LIN {X 0,Y 260.477,Z 576.066,A -85,B 0,C 180,E1 -18837.737,E2 -18837.737} C_VEL
LIN {X 0,Y 264.246,Z 563.841,A -85,B 0,C 180,E1 -18840.132,E2 -18840.132} C_VEL
LIN {X 0,Y 267.827,Z 551.379,A -85,B 0,C 180,E1 -18842.097,E2 -18842.097} C_VEL
LIN {X 0,Y 271.196,Z 538.149,A -85,B 0,C 180,E1 -18843.781,E2 -18843.781} C_VEL
LIN {X 0,Y 274.264,Z 524.044,A -85,B 0,C 180,E1 -18845.208,E2 -18845.208} C_VEL
LIN {X 0,Y 276.82,Z 510.254,A -85,B 0,C 180,E1 -18846.288,E2 -18846.288} C_VEL
LIN {X 0,Y 279.114,Z 494.819,A -85,B 0,C 180,E1 -18847.178,E2 -18847.178} C_VEL
LIN {X 0,Y 280.649,Z 479.547,A -85,B 0,C 180,E1 -18847.787,E2 -18847.787} C_VEL
LIN {X 0,Y 285.626,Z 378.515,A -85,B 0,C 180,E1 -18850.247,E2 -18850.247} C_VEL
LIN {X 0,Y 285.487,Z 376.742,A -85,B 0,C 180,E1 -18850.327,E2 -18850.327} C_VEL
LIN {X 0,Y 278.337,Z 360.16,A -85,B 0,C 180,E1 -18852.139,E2 -18852.139} C_VEL
LIN {X 0,Y 270.765,Z 345.131,A -85,B 0,C 180,E1 -18854.134,E2 -18854.134} C_VEL
LIN {X 0,Y 263.382,Z 332.001,A -85,B 0,C 180,E1 -18856.203,E2 -18856.203} C_VEL
LIN {X 0,Y 256.795,Z 321.549,A -85,B 0,C 180,E1 -18858.171,E2 -18858.171} C_VEL
LIN {X 0,Y 253.581,Z 316.573,A -85,B 0,C 180,E1 -18859.193,E2 -18859.193} C_VEL
LIN {X 0,Y 250.484,Z 311.706,A -85,B 0,C 180,E1 -18860.269,E2 -18860.269} C_VEL
LIN {X 0,Y 249.039,Z 307.085,A -85,B 0,C 180,E1 -18862.618,E2 -18862.618} C_VEL
LIN {X 0,Y 249.037,Z 307.088,A -85,B 0,C 180,E1 -18865.639,E2 -18865.639} C_VEL
LIN {X 0,Y 248.994,Z 307.089,A -85,B 0,C 180,E1 -18869.465,E2 -18869.465} C_VEL
LIN {X 0,Y 249.008,Z 307.086,A -85,B 0,C 180,E1 -18873.155,E2 -18873.155} C_VEL
LIN {X 0,Y 248.998,Z 307.089,A -85,B 0,C 180,E1 -18876.725,E2 -18876.725} C_VEL
LIN {X 0,Y 249.038,Z 307.057,A -85,B 0,C 180,E1 -18880.206,E2 -18880.206} C_VEL
LIN {X 0,Y 249.151,Z 307.067,A -85,B 0,C 180,E1 -18883.616,E2 -18883.616} C_VEL
LIN {X 0,Y 249.177,Z 307.04,A -85,B 0,C 180,E1 -18886.96,E2 -18886.96} C_VEL
LIN {X 0,Y 249.365,Z 307.025,A -85,B 0,C 180,E1 -18890.538,E2 -18890.538} C_VEL
LIN {X 0,Y 249.415,Z 307.035,A -85,B 0,C 180,E1 -18893.529,E2 -18893.529} C_VEL
LIN {X 0,Y 249.653,Z 307.001,A -85,B 0,C 180,E1 -18898.387,E2 -18898.387} C_VEL
LIN {X 0,Y 249.65,Z 307.007,A -85,B 0,C 180,E1 -18901.613,E2 -18901.613} C_VEL
LIN {X 0,Y 249.416,Z 307.032,A -85,B 0,C 180,E1 -18906.679,E2 -18906.679} C_VEL
LIN {X 0,Y 249.326,Z 307.05,A -85,B 0,C 180,E1 -18909.737,E2 -18909.737} C_VEL
LIN {X 0,Y 249.164,Z 307.065,A -85,B 0,C 180,E1 -18914.706,E2 -18914.706} C_VEL
LIN {X 0,Y 249.088,Z 307.072,A -85,B 0,C 180,E1 -18918.081,E2 -18918.081} C_VEL
LIN {X 0,Y 249.041,Z 307.055,A -85,B 0,C 180,E1 -18921.523,E2 -18921.523} C_VEL
LIN {X 0,Y 249.107,Z 307.067,A -85,B 0,C 180,E1 -18925.474,E2 -18925.474} C_VEL
LIN {X 0,Y 249.058,Z 307.066,A -85,B 0,C 180,E1 -18928.986,E2 -18928.986} C_VEL
LIN {X 0,Y 249.026,Z 307.084,A -85,B 0,C 180,E1 -18932.427,E2 -18932.427} C_VEL
LIN {X 0,Y 249.043,Z 307.088,A -85,B 0,C 180,E1 -18936.343,E2 -18936.343} C_VEL
LIN {X 0,Y 249.022,Z 307.166,A -85,B 0,C 180,E1 -18939.617,E2 -18939.617} C_VEL
LIN {X 0,Y 249.906,Z 309.755,A -85,B 0,C 180,E1 -18939.977,E2 -18939.977} C_VEL
LIN {X 0,Y 251.813,Z 311.92,A -85,B 0,C 180,E1 -18940.59,E2 -18940.59} C_VEL
LIN {X 0,Y 252.602,Z 312.645,A -85,B 0,C 180,E1 -18940.831,E2 -18940.831} C_VEL
LIN {X 0,Y 254.745,Z 315.993,A -85,B 0,C 180,E1 -18941.53,E2 -18941.53} C_VEL
LIN {X 0,Y 256.163,Z 317.683,A -85,B 0,C 180,E1 -18941.96,E2 -18941.96} C_VEL
LIN {X 0,Y 258.928,Z 321.433,A -85,B 0,C 180,E1 -18942.792,E2 -18942.792} C_VEL
LIN {X 0,Y 268.098,Z 334.977,A -85,B 0,C 180,E1 -18945.388,E2 -18945.388} C_VEL
LIN {X 0,Y 274.88,Z 345.917,A -85,B 0,C 180,E1 -18947.161,E2 -18947.161} C_VEL
LIN {X 0,Y 281.793,Z 359.713,A -85,B 0,C 180,E1 -18948.921,E2 -18948.921} C_VEL
LIN {X 0,Y 285.944,Z 368.841,A -85,B 0,C 180,E1 -18949.943,E2 -18949.943} C_VEL
LIN {X 0,Y 281.179,Z 467.093,A -85,B 0,C 180,E1 -18952.353,E2 -18952.353} C_VEL
LIN {X 0,Y 279.682,Z 482.247,A -85,B 0,C 180,E1 -18952.967,E2 -18952.967} C_VEL
LIN {X 0,Y 277.739,Z 496.979,A -85,B 0,C 180,E1 -18953.851,E2 -18953.851} C_VEL
LIN {X 0,Y 275.33,Z 511.361,A -85,B 0,C 180,E1 -18955.013,E2 -18955.013} C_VEL
LIN {X 0,Y 272.275,Z 525.892,A -85,B 0,C 180,E1 -18956.515,E2 -18956.515} C_VEL
LIN {X 0,Y 269.174,Z 538.098,A -85,B 0,C 180,E1 -18958.082,E2 -18958.082} C_VEL
LIN {X 0,Y 266.055,Z 549.441,A -85,B 0,C 180,E1 -18959.875,E2 -18959.875} C_VEL
LIN {X 0,Y 262.464,Z 561.007,A -85,B 0,C 180,E1 -18962.085,E2 -18962.085} C_VEL
LIN {X 0,Y 259.548,Z 570.521,A -85,B 0,C 180,E1 -18964.327,E2 -18964.327} C_VEL
LIN {X 0,Y 256.366,Z 579.961,A -85,B 0,C 180,E1 -18967.006,E2 -18967.006} C_VEL
LIN {X 0,Y 253.642,Z 587.816,A -85,B 0,C 180,E1 -18969.736,E2 -18969.736} C_VEL
LIN {X 0,Y 251.256,Z 595.141,A -85,B 0,C 180,E1 -18972.921,E2 -18972.921} C_VEL
LIN {X 0,Y 249.39,Z 600.95,A -85,B 0,C 180,E1 -18976.141,E2 -18976.141} C_VEL
LIN {X 0,Y 248.47,Z 604.384,A -85,B 0,C 180,E1 -18978.581,E2 -18978.581} C_VEL
LIN {X 0,Y 247.638,Z 607.86,A -85,B 0,C 180,E1 -18981.842,E2 -18981.842} C_VEL
LIN {X 0,Y 247.134,Z 610.155,A -85,B 0,C 180,E1 -18985.106,E2 -18985.106} C_VEL
LIN {X 0,Y 246.995,Z 611.323,A -85,B 0,C 180,E1 -18988.37,E2 -18988.37} C_VEL
LIN {X 0,Y 246.994,Z 611.336,A -85,B 0,C 180,E1 -18991.63,E2 -18991.63} C_VEL
LIN {X 0,Y 247.128,Z 610.22,A -85,B 0,C 180,E1 -18994.894,E2 -18994.894} C_VEL
LIN {X 0,Y 247.576,Z 607.975,A -85,B 0,C 180,E1 -18998.16,E2 -18998.16} C_VEL
LIN {X 0,Y 248.443,Z 604.544,A -85,B 0,C 180,E1 -19001.421,E2 -19001.421} C_VEL
LIN {X 0,Y 249.783,Z 599.845,A -85,B 0,C 180,E1 -19004.668,E2 -19004.668} C_VEL
LIN {X 0,Y 251.755,Z 593.749,A -85,B 0,C 180,E1 -19007.883,E2 -19007.883} C_VEL
LIN {X 0,Y 254.327,Z 586.069,A -85,B 0,C 180,E1 -19011.053,E2 -19011.053} C_VEL
LIN {X 0,Y 257.145,Z 577.876,A -85,B 0,C 180,E1 -19013.773,E2 -19013.773} C_VEL
LIN {X 0,Y 260.504,Z 567.999,A -85,B 0,C 180,E1 -19016.432,E2 -19016.432} C_VEL
LIN {X 0,Y 263.554,Z 557.877,A -85,B 0,C 180,E1 -19018.684,E2 -19018.684} C_VEL
LIN {X 0,Y 267.19,Z 545.809,A -85,B 0,C 180,E1 -19020.857,E2 -19020.857} C_VEL
LIN {X 0,Y 270.434,Z 533.706,A -85,B 0,C 180,E1 -19022.631,E2 -19022.631} C_VEL
LIN {X 0,Y 273.51,Z 520.55,A -85,B 0,C 180,E1 -19024.199,E2 -19024.199} C_VEL
LIN {X 0,Y 276.065,Z 507.506,A -85,B 0,C 180,E1 -19025.447,E2 -19025.447} C_VEL
LIN {X 0,Y 278.318,Z 493.311,A -85,B 0,C 180,E1 -19026.511,E2 -19026.511} C_VEL
LIN {X 0,Y 280.218,Z 478.014,A -85,B 0,C 180,E1 -19027.345,E2 -19027.345} C_VEL
LIN {X 0,Y 281.501,Z 463.213,A -85,B 0,C 180,E1 -19027.879,E2 -19027.879} C_VEL
LIN {X 0,Y 286.04,Z 368.931,A -85,B 0,C 180,E1 -19030.172,E2 -19030.172} C_VEL
LIN {X 0,Y 278.222,Z 352.196,A -85,B 0,C 180,E1 -19032.124,E2 -19032.124} C_VEL
LIN {X 0,Y 273.365,Z 343.191,A -85,B 0,C 180,E1 -19033.376,E2 -19033.376} C_VEL
LIN {X 0,Y 265.536,Z 331.06,A -85,B 0,C 180,E1 -19035.462,E2 -19035.462} C_VEL
LIN {X 0,Y 258.345,Z 320.791,A -85,B 0,C 180,E1 -19037.531,E2 -19037.531} C_VEL
LIN {X 0,Y 255.483,Z 316.712,A -85,B 0,C 180,E1 -19038.412,E2 -19038.412} C_VEL
LIN {X 0,Y 253.02,Z 313.492,A -85,B 0,C 180,E1 -19039.185,E2 -19039.185} C_VEL
LIN {X 0,Y 252.146,Z 312.144,A -85,B 0,C 180,E1 -19039.475,E2 -19039.475} C_VEL
LIN {X 0,Y 250.089,Z 310.064,A -85,B 0,C 180,E1 -19040.125,E2 -19040.125} C_VEL
LIN {X 0,Y 249.079,Z 307.384,A -85,B 0,C 180,E1 -19040.525,E2 -19040.525} C_VEL
LIN {X 0,Y 249.015,Z 307.093,A -85,B 0,C 180,E1 -19040.578,E2 -19040.578} C_VEL
LIN {X 0,Y 249.039,Z 307.073,A -85,B 0,C 180,E1 -19044.922,E2 -19044.922} C_VEL
LIN {X 0,Y 249.001,Z 307.059,A -85,B 0,C 180,E1 -19049.466,E2 -19049.466} C_VEL
LIN {X 0,Y 249.053,Z 307.086,A -85,B 0,C 180,E1 -19053.16,E2 -19053.16} C_VEL
LIN {X 0,Y 249.052,Z 307.087,A -85,B 0,C 180,E1 -19056.73,E2 -19056.73} C_VEL
LIN {X 0,Y 249.077,Z 307.084,A -85,B 0,C 180,E1 -19060.209,E2 -19060.209} C_VEL
LIN {X 0,Y 249.097,Z 307.071,A -85,B 0,C 180,E1 -19061.859,E2 -19061.859} C_VEL
LIN {X 0,Y 248.501,Z 307.151,A -85,B 0,C 180,E1 -19063.21,E2 -19063.21} C_VEL
LIN {X 0,Y 245.667,Z 307.506,A -85,B 0,C 180,E1 -19065.413,E2 -19065.413} C_VEL
LIN {X 0,Y 243.243,Z 307.808,A -85,B 0,C 180,E1 -19067.207,E2 -19067.207} C_VEL
LIN {X 0,Y 242.239,Z 307.936,A -85,B 0,C 180,E1 -19068.6,E2 -19068.6} C_VEL
LIN {X 0,Y 242.18,Z 307.936,A -85,B 0,C 180,E1 -19069.072,E2 -19069.072} C_VEL
LIN {X 0,Y 242.382,Z 307.907,A -85,B 0,C 180,E1 -19071.664,E2 -19071.664} C_VEL
LIN {X 0,Y 242.226,Z 307.925,A -85,B 0,C 180,E1 -19075.006,E2 -19075.006} C_VEL
LIN {X 0,Y 242.617,Z 307.888,A -85,B 0,C 180,E1 -19078.34,E2 -19078.34} C_VEL
LIN {X 0,Y 242.613,Z 307.887,A -85,B 0,C 180,E1 -19081.66,E2 -19081.66} C_VEL
LIN {X 0,Y 242.397,Z 307.917,A -85,B 0,C 180,E1 -19086.66,E2 -19086.66} C_VEL
LIN {X 0,Y 242.259,Z 307.925,A -85,B 0,C 180,E1 -19090.024,E2 -19090.024} C_VEL
LIN {X 0,Y 242.114,Z 307.952,A -85,B 0,C 180,E1 -19095.144,E2 -19095.144} C_VEL
LIN {X 0,Y 242.024,Z 307.956,A -85,B 0,C 180,E1 -19098.628,E2 -19098.628} C_VEL
LIN {X 0,Y 241.967,Z 307.961,A -85,B 0,C 180,E1 -19102.184,E2 -19102.184} C_VEL
LIN {X 0,Y 241.981,Z 307.959,A -85,B 0,C 180,E1 -19105.827,E2 -19105.827} C_VEL
LIN {X 0,Y 241.962,Z 307.972,A -85,B 0,C 180,E1 -19109.589,E2 -19109.589} C_VEL
LIN {X 0,Y 241.974,Z 307.959,A -85,B 0,C 180,E1 -19113.493,E2 -19113.493} C_VEL
LIN {X 0,Y 241.998,Z 308.143,A -85,B 0,C 180,E1 -19115.739,E2 -19115.739} C_VEL
LIN {X 0,Y 243.266,Z 311.805,A -85,B 0,C 180,E1 -19117.623,E2 -19117.623} C_VEL
LIN {X 0,Y 246.159,Z 316.163,A -85,B 0,C 180,E1 -19118.682,E2 -19118.682} C_VEL
LIN {X 0,Y 248.289,Z 319.312,A -85,B 0,C 180,E1 -19119.428,E2 -19119.428} C_VEL
LIN {X 0,Y 251.893,Z 324.806,A -85,B 0,C 180,E1 -19120.644,E2 -19120.644} C_VEL
LIN {X 0,Y 257.896,Z 334.42,A -85,B 0,C 180,E1 -19122.552,E2 -19122.552} C_VEL
LIN {X 0,Y 265.153,Z 347.057,A -85,B 0,C 180,E1 -19124.701,E2 -19124.701} C_VEL
LIN {X 0,Y 272.745,Z 362.134,A -85,B 0,C 180,E1 -19126.815,E2 -19126.815} C_VEL
LIN {X 0,Y 279.117,Z 376.624,A -85,B 0,C 180,E1 -19128.511,E2 -19128.511} C_VEL
LIN {X 0,Y 280.222,Z 379.318,A -85,B 0,C 180,E1 -19128.799,E2 -19128.799} C_VEL
LIN {X 0,Y 275.522,Z 474.523,A -85,B 0,C 180,E1 -19131.148,E2 -19131.148} C_VEL
LIN {X 0,Y 274.146,Z 489.815,A -85,B 0,C 180,E1 -19131.68,E2 -19131.68} C_VEL
LIN {X 0,Y 271.984,Z 505.365,A -85,B 0,C 180,E1 -19132.495,E2 -19132.495} C_VEL
LIN {X 0,Y 269.297,Z 520.239,A -85,B 0,C 180,E1 -19133.58,E2 -19133.58} C_VEL
LIN {X 0,Y 266.114,Z 534.597,A -85,B 0,C 180,E1 -19134.955,E2 -19134.955} C_VEL
LIN {X 0,Y 262.902,Z 547.521,A -85,B 0,C 180,E1 -19136.541,E2 -19136.541} C_VEL
LIN {X 0,Y 259.416,Z 559.534,A -85,B 0,C 180,E1 -19138.339,E2 -19138.339} C_VEL
LIN {X 0,Y 255.899,Z 570.666,A -85,B 0,C 180,E1 -19140.374,E2 -19140.374} C_VEL
LIN {X 0,Y 252.446,Z 581.236,A -85,B 0,C 180,E1 -19142.745,E2 -19142.745} C_VEL
LIN {X 0,Y 249.249,Z 590.949,A -85,B 0,C 180,E1 -19145.425,E2 -19145.425} C_VEL
LIN {X 0,Y 246.294,Z 599.278,A -85,B 0,C 180,E1 -19148.226,E2 -19148.226} C_VEL
LIN {X 0,Y 243.714,Z 607.112,A -85,B 0,C 180,E1 -19151.506,E2 -19151.506} C_VEL
LIN {X 0,Y 241.837,Z 613.352,A -85,B 0,C 180,E1 -19154.839,E2 -19154.839} C_VEL
LIN {X 0,Y 240.593,Z 618.183,A -85,B 0,C 180,E1 -19158.201,E2 -19158.201} C_VEL
LIN {X 0,Y 239.985,Z 621.73,A -85,B 0,C 180,E1 -19161.58,E2 -19161.58} C_VEL
LIN {X 0,Y 239.765,Z 624.067,A -85,B 0,C 180,E1 -19164.955,E2 -19164.955} C_VEL
LIN {X 0,Y 239.829,Z 625.244,A -85,B 0,C 180,E1 -19168.321,E2 -19168.321} C_VEL
LIN {X 0,Y 239.89,Z 625.4,A -85,B 0,C 180,E1 -19170,E2 -19170} C_VEL
LIN {X 0,Y 239.744,Z 624.785,A -85,B 0,C 180,E1 -19173.361,E2 -19173.361} C_VEL
LIN {X 0,Y 239.785,Z 623.015,A -85,B 0,C 180,E1 -19176.733,E2 -19176.733} C_VEL
LIN {X 0,Y 240.229,Z 620.071,A -85,B 0,C 180,E1 -19180.109,E2 -19180.109} C_VEL
LIN {X 0,Y 241.167,Z 615.885,A -85,B 0,C 180,E1 -19183.481,E2 -19183.481} C_VEL
LIN {X 0,Y 242.591,Z 610.344,A -85,B 0,C 180,E1 -19186.84,E2 -19186.84} C_VEL
LIN {X 0,Y 244.896,Z 603.312,A -85,B 0,C 180,E1 -19190.143,E2 -19190.143} C_VEL
LIN {X 0,Y 247.899,Z 594.571,A -85,B 0,C 180,E1 -19193.384,E2 -19193.384} C_VEL
LIN {X 0,Y 250.555,Z 586.782,A -85,B 0,C 180,E1 -19195.756,E2 -19195.756} C_VEL
LIN {X 0,Y 254.146,Z 575.858,A -85,B 0,C 180,E1 -19198.49,E2 -19198.49} C_VEL
LIN {X 0,Y 258.103,Z 563.634,A -85,B 0,C 180,E1 -19200.927,E2 -19200.927} C_VEL
LIN {X 0,Y 261.445,Z 552.4,A -85,B 0,C 180,E1 -19202.75,E2 -19202.75} C_VEL
LIN {X 0,Y 265.107,Z 538.703,A -85,B 0,C 180,E1 -19204.55,E2 -19204.55} C_VEL
LIN {X 0,Y 268.472,Z 523.834,A -85,B 0,C 180,E1 -19206.085,E2 -19206.085} C_VEL
LIN {X 0,Y 271.143,Z 510.044,A -85,B 0,C 180,E1 -19207.174,E2 -19207.174} C_VEL
LIN {X 0,Y 273.5,Z 494.607,A -85,B 0,C 180,E1 -19208.075,E2 -19208.075} C_VEL
LIN {X 0,Y 275.067,Z 479.328,A -85,B 0,C 180,E1 -19208.694,E2 -19208.694} C_VEL
LIN {X 0,Y 279.58,Z 391.475,A -85,B 0,C 180,E1 -19210.864,E2 -19210.864} C_VEL
LIN {X 0,Y 280.114,Z 379.234,A -85,B 0,C 180,E1 -19211.176,E2 -19211.176} C_VEL
LIN {X 0,Y 273.524,Z 363.866,A -85,B 0,C 180,E1 -19212.921,E2 -19212.921} C_VEL
LIN {X 0,Y 266.605,Z 349.897,A -85,B 0,C 180,E1 -19214.824,E2 -19214.824} C_VEL
LIN {X 0,Y 259.318,Z 336.779,A -85,B 0,C 180,E1 -19216.951,E2 -19216.951} C_VEL
LIN {X 0,Y 253.151,Z 326.806,A -85,B 0,C 180,E1 -19218.873,E2 -19218.873} C_VEL
LIN {X 0,Y 249.75,Z 321.507,A -85,B 0,C 180,E1 -19219.997,E2 -19219.997} C_VEL
LIN {X 0,Y 246.292,Z 316.344,A -85,B 0,C 180,E1 -19221.192,E2 -19221.192} C_VEL
LIN {X 0,Y 243.196,Z 311.686,A -85,B 0,C 180,E1 -19222.319,E2 -19222.319} C_VEL
LIN {X 0,Y 241.981,Z 307.961,A -85,B 0,C 180,E1 -19224.374,E2 -19224.374} C_VEL
LIN {X 0,Y 241.947,Z 307.972,A -85,B 0,C 180,E1 -19228.476,E2 -19228.476} C_VEL
LIN {X 0,Y 241.949,Z 307.967,A -85,B 0,C 180,E1 -19232.306,E2 -19232.306} C_VEL
LIN {X 0,Y 241.95,Z 307.965,A -85,B 0,C 180,E1 -19236.005,E2 -19236.005} C_VEL
LIN {X 0,Y 241.977,Z 307.942,A -85,B 0,C 180,E1 -19239.603,E2 -19239.603} C_VEL
LIN {X 0,Y 242.107,Z 307.938,A -85,B 0,C 180,E1 -19243.318,E2 -19243.318} C_VEL
LIN {X 0,Y 242.153,Z 307.903,A -85,B 0,C 180,E1 -19248.278,E2 -19248.278} C_VEL
LIN {X 0,Y 242.351,Z 307.918,A -85,B 0,C 180,E1 -19251.663,E2 -19251.663} C_VEL
LIN {X 0,Y 242.384,Z 307.912,A -85,B 0,C 180,E1 -19253.34,E2 -19253.34} C_VEL
LIN {X 0,Y 242.612,Z 307.878,A -85,B 0,C 180,E1 -19258.34,E2 -19258.34} C_VEL
LIN {X 0,Y 242.611,Z 307.884,A -85,B 0,C 180,E1 -19261.66,E2 -19261.66} C_VEL
LIN {X 0,Y 242.398,Z 307.906,A -85,B 0,C 180,E1 -19266.66,E2 -19266.66} C_VEL
LIN {X 0,Y 242.254,Z 307.928,A -85,B 0,C 180,E1 -19270.024,E2 -19270.024} C_VEL
LIN {X 0,Y 242.114,Z 307.942,A -85,B 0,C 180,E1 -19275.144,E2 -19275.144} C_VEL
LIN {X 0,Y 242.025,Z 307.941,A -85,B 0,C 180,E1 -19278.628,E2 -19278.628} C_VEL
LIN {X 0,Y 241.983,Z 307.941,A -85,B 0,C 180,E1 -19282.183,E2 -19282.183} C_VEL
LIN {X 0,Y 242.045,Z 307.939,A -85,B 0,C 180,E1 -19285.83,E2 -19285.83} C_VEL
LIN {X 0,Y 241.999,Z 307.955,A -85,B 0,C 180,E1 -19289.585,E2 -19289.585} C_VEL
LIN {X 0,Y 241.976,Z 307.969,A -85,B 0,C 180,E1 -19293.494,E2 -19293.494} C_VEL
LIN {X 0,Y 241.988,Z 307.983,A -85,B 0,C 180,E1 -19297.582,E2 -19297.582} C_VEL
LIN {X 0,Y 242.936,Z 310.696,A -85,B 0,C 180,E1 -19298.003,E2 -19298.003} C_VEL
LIN {X 0,Y 244.853,Z 312.841,A -85,B 0,C 180,E1 -19298.677,E2 -19298.677} C_VEL
LIN {X 0,Y 245.764,Z 313.765,A -85,B 0,C 180,E1 -19298.986,E2 -19298.986} C_VEL
LIN {X 0,Y 248.012,Z 317.166,A -85,B 0,C 180,E1 -19299.78,E2 -19299.78} C_VEL
LIN {X 0,Y 249.476,Z 318.808,A -85,B 0,C 180,E1 -19300.257,E2 -19300.257} C_VEL
LIN {X 0,Y 252.072,Z 322.342,A -85,B 0,C 180,E1 -19301.105,E2 -19301.105} C_VEL
LIN {X 0,Y 259.349,Z 332.783,A -85,B 0,C 180,E1 -19303.345,E2 -19303.345} C_VEL
LIN {X 0,Y 267.478,Z 345.207,A -85,B 0,C 180,E1 -19305.635,E2 -19305.635} C_VEL
LIN {X 0,Y 272.335,Z 353.843,A -85,B 0,C 180,E1 -19306.941,E2 -19306.941} C_VEL
LIN {X 0,Y 279.378,Z 368.706,A -85,B 0,C 180,E1 -19308.787,E2 -19308.787} C_VEL
LIN {X 0,Y 280.44,Z 371.158,A -85,B 0,C 180,E1 -19309.06,E2 -19309.06} C_VEL
LIN {X 0,Y 275.6,Z 467.311,A -85,B 0,C 180,E1 -19311.453,E2 -19311.453} C_VEL
LIN {X 0,Y 274.062,Z 482.461,A -85,B 0,C 180,E1 -19312.075,E2 -19312.075} C_VEL
LIN {X 0,Y 272.049,Z 497.19,A -85,B 0,C 180,E1 -19312.97,E2 -19312.97} C_VEL
LIN {X 0,Y 269.74,Z 510.156,A -85,B 0,C 180,E1 -19314.013,E2 -19314.013} C_VEL
LIN {X 0,Y 266.756,Z 524.548,A -85,B 0,C 180,E1 -19315.499,E2 -19315.499} C_VEL
LIN {X 0,Y 263.514,Z 537.018,A -85,B 0,C 180,E1 -19317.085,E2 -19317.085} C_VEL
LIN {X 0,Y 260.264,Z 548.583,A -85,B 0,C 180,E1 -19318.907,E2 -19318.907} C_VEL
LIN {X 0,Y 256.47,Z 560.443,A -85,B 0,C 180,E1 -19321.179,E2 -19321.179} C_VEL
LIN {X 0,Y 253.169,Z 570.727,A -85,B 0,C 180,E1 -19323.631,E2 -19323.631} C_VEL
LIN {X 0,Y 249.834,Z 580.166,A -85,B 0,C 180,E1 -19326.369,E2 -19326.369} C_VEL
LIN {X 0,Y 246.978,Z 588.021,A -85,B 0,C 180,E1 -19329.164,E2 -19329.164} C_VEL
LIN {X 0,Y 244.438,Z 595.347,A -85,B 0,C 180,E1 -19332.429,E2 -19332.429} C_VEL
LIN {X 0,Y 242.477,Z 601.155,A -85,B 0,C 180,E1 -19335.738,E2 -19335.738} C_VEL
LIN {X 0,Y 241.5,Z 604.589,A -85,B 0,C 180,E1 -19338.246,E2 -19338.246} C_VEL
LIN {X 0,Y 240.61,Z 608.063,A -85,B 0,C 180,E1 -19341.602,E2 -19341.602} C_VEL
LIN {X 0,Y 240.058,Z 610.359,A -85,B 0,C 180,E1 -19344.961,E2 -19344.961} C_VEL
LIN {X 0,Y 239.907,Z 611.526,A -85,B 0,C 180,E1 -19348.321,E2 -19348.321} C_VEL
LIN {X 0,Y 239.906,Z 611.538,A -85,B 0,C 180,E1 -19351.679,E2 -19351.679} C_VEL
LIN {X 0,Y 240.058,Z 610.423,A -85,B 0,C 180,E1 -19355.039,E2 -19355.039} C_VEL
LIN {X 0,Y 240.523,Z 608.178,A -85,B 0,C 180,E1 -19358.401,E2 -19358.401} C_VEL
LIN {X 0,Y 241.458,Z 604.747,A -85,B 0,C 180,E1 -19361.756,E2 -19361.756} C_VEL
LIN {X 0,Y 242.906,Z 600.047,A -85,B 0,C 180,E1 -19365.093,E2 -19365.093} C_VEL
LIN {X 0,Y 244.989,Z 593.951,A -85,B 0,C 180,E1 -19368.394,E2 -19368.394} C_VEL
LIN {X 0,Y 247.669,Z 586.272,A -85,B 0,C 180,E1 -19371.647,E2 -19371.647} C_VEL
LIN {X 0,Y 250.646,Z 578.077,A -85,B 0,C 180,E1 -19374.429,E2 -19374.429} C_VEL
LIN {X 0,Y 254.129,Z 568.2,A -85,B 0,C 180,E1 -19377.149,E2 -19377.149} C_VEL
LIN {X 0,Y 257.328,Z 558.077,A -85,B 0,C 180,E1 -19379.445,E2 -19379.445} C_VEL
LIN {X 0,Y 261.127,Z 546.009,A -85,B 0,C 180,E1 -19381.656,E2 -19381.656} C_VEL
LIN {X 0,Y 264.492,Z 533.905,A -85,B 0,C 180,E1 -19383.459,E2 -19383.459} C_VEL
LIN {X 0,Y 267.666,Z 520.748,A -85,B 0,C 180,E1 -19385.054,E2 -19385.054} C_VEL
LIN {X 0,Y 270.175,Z 508.445,A -85,B 0,C 180,E1 -19386.255,E2 -19386.255} C_VEL
LIN {X 0,Y 272.475,Z 494.803,A -85,B 0,C 180,E1 -19387.31,E2 -19387.31} C_VEL
LIN {X 0,Y 274.44,Z 480.03,A -85,B 0,C 180,E1 -19388.155,E2 -19388.155} C_VEL
LIN {X 0,Y 275.86,Z 464.898,A -85,B 0,C 180,E1 -19388.738,E2 -19388.738} C_VEL
LIN {X 0,Y 280.557,Z 372.002,A -85,B 0,C 180,E1 -19391.028,E2 -19391.028} C_VEL
LIN {X 0,Y 280.254,Z 370.496,A -85,B 0,C 180,E1 -19391.132,E2 -19391.132} C_VEL
LIN {X 0,Y 272.656,Z 354.369,A -85,B 0,C 180,E1 -19393.12,E2 -19393.12} C_VEL
LIN {X 0,Y 267.696,Z 345.456,A -85,B 0,C 180,E1 -19394.457,E2 -19394.457} C_VEL
LIN {X 0,Y 258.168,Z 330.912,A -85,B 0,C 180,E1 -19397.166,E2 -19397.166} C_VEL
LIN {X 0,Y 251.797,Z 322.034,A -85,B 0,C 180,E1 -19399.143,E2 -19399.143} C_VEL
LIN {X 0,Y 248.627,Z 317.741,A -85,B 0,C 180,E1 -19400.19,E2 -19400.19} C_VEL
LIN {X 0,Y 246.371,Z 314.945,A -85,B 0,C 180,E1 -19400.955,E2 -19400.955} C_VEL
LIN {X 0,Y 245.408,Z 313.2,A -85,B 0,C 180,E1 -19401.315,E2 -19401.315} C_VEL
LIN {X 0,Y 243.172,Z 311.084,A -85,B 0,C 180,E1 -19402.082,E2 -19402.082} C_VEL
LIN {X 0,Y 242.041,Z 308.398,A -85,B 0,C 180,E1 -19402.558,E2 -19402.558} C_VEL
LIN {X 0,Y 241.972,Z 307.943,A -85,B 0,C 180,E1 -19402.677,E2 -19402.677} C_VEL
LIN {X 0,Y 241.983,Z 307.95,A -85,B 0,C 180,E1 -19407.377,E2 -19407.377} C_VEL
LIN {X 0,Y 241.98,Z 307.94,A -85,B 0,C 180,E1 -19410.608,E2 -19410.608} C_VEL
LIN {X 0,Y 242.045,Z 307.951,A -85,B 0,C 180,E1 -19414.18,E2 -19414.18} C_VEL
LIN {X 0,Y 242.017,Z 307.953,A -85,B 0,C 180,E1 -19418.315,E2 -19418.315} C_VEL
LIN {X 0,Y 242.11,Z 307.945,A -85,B 0,C 180,E1 -19423.316,E2 -19423.316} C_VEL
LIN {X 0,Y 242.16,Z 307.944,A -85,B 0,C 180,E1 -19428.278,E2 -19428.278} C_VEL
LIN {X 0,Y 242.18,Z 307.936,A -85,B 0,C 180,E1 -19429.072,E2 -19429.072} C_VEL
LIN {X 0,Y 241.556,Z 308.014,A -85,B 0,C 180,E1 -19430.461,E2 -19430.461} C_VEL
LIN {X 0,Y 238.684,Z 308.376,A -85,B 0,C 180,E1 -19432.726,E2 -19432.726} C_VEL
LIN {X 0,Y 236.264,Z 308.671,A -85,B 0,C 180,E1 -19434.573,E2 -19434.573} C_VEL
LIN {X 0,Y 235.3,Z 308.787,A -85,B 0,C 180,E1 -19436.007,E2 -19436.007} C_VEL
LIN {X 0,Y 235.263,Z 308.795,A -85,B 0,C 180,E1 -19436.492,E2 -19436.492} C_VEL
LIN {X 0,Y 235.575,Z 308.765,A -85,B 0,C 180,E1 -19438.29,E2 -19438.29} C_VEL
LIN {X 0,Y 235.571,Z 308.764,A -85,B 0,C 180,E1 -19441.709,E2 -19441.709} C_VEL
LIN {X 0,Y 235.349,Z 308.796,A -85,B 0,C 180,E1 -19446.86,E2 -19446.86} C_VEL
LIN {X 0,Y 235.205,Z 308.806,A -85,B 0,C 180,E1 -19450.328,E2 -19450.328} C_VEL
LIN {X 0,Y 235.063,Z 308.833,A -85,B 0,C 180,E1 -19455.61,E2 -19455.61} C_VEL
LIN {X 0,Y 234.962,Z 308.841,A -85,B 0,C 180,E1 -19459.209,E2 -19459.209} C_VEL
LIN {X 0,Y 234.911,Z 308.843,A -85,B 0,C 180,E1 -19462.888,E2 -19462.888} C_VEL
LIN {X 0,Y 234.92,Z 308.841,A -85,B 0,C 180,E1 -19466.663,E2 -19466.663} C_VEL
LIN {X 0,Y 234.893,Z 308.85,A -85,B 0,C 180,E1 -19470.573,E2 -19470.573} C_VEL
LIN {X 0,Y 234.922,Z 308.87,A -85,B 0,C 180,E1 -19473.796,E2 -19473.796} C_VEL
LIN {X 0,Y 235.779,Z 311.451,A -85,B 0,C 180,E1 -19475.193,E2 -19475.193} C_VEL
LIN {X 0,Y 239.087,Z 316.219,A -85,B 0,C 180,E1 -19476.53,E2 -19476.53} C_VEL
LIN {X 0,Y 240.589,Z 318.413,A -85,B 0,C 180,E1 -19477.114,E2 -19477.114} C_VEL
LIN {X 0,Y 244.451,Z 323.947,A -85,B 0,C 180,E1 -19478.542,E2 -19478.542} C_VEL
LIN {X 0,Y 250.937,Z 334.155,A -85,B 0,C 180,E1 -19480.792,E2 -19480.792} C_VEL
LIN {X 0,Y 257.446,Z 345.26,A -85,B 0,C 180,E1 -19482.88,E2 -19482.88} C_VEL
LIN {X 0,Y 264.059,Z 357.687,A -85,B 0,C 180,E1 -19484.864,E2 -19484.864} C_VEL
LIN {X 0,Y 270.74,Z 371.812,A -85,B 0,C 180,E1 -19486.763,E2 -19486.763} C_VEL
LIN {X 0,Y 274.78,Z 381.476,A -85,B 0,C 180,E1 -19487.879,E2 -19487.879} C_VEL
LIN {X 0,Y 270.024,Z 474.338,A -85,B 0,C 180,E1 -19490.201,E2 -19490.201} C_VEL
LIN {X 0,Y 268.609,Z 489.623,A -85,B 0,C 180,E1 -19490.74,E2 -19490.74} C_VEL
LIN {X 0,Y 266.399,Z 505.17,A -85,B 0,C 180,E1 -19491.567,E2 -19491.567} C_VEL
LIN {X 0,Y 263.626,Z 520.043,A -85,B 0,C 180,E1 -19492.665,E2 -19492.665} C_VEL
LIN {X 0,Y 260.231,Z 534.723,A -85,B 0,C 180,E1 -19494.09,E2 -19494.09} C_VEL
LIN {X 0,Y 256.626,Z 548.616,A -85,B 0,C 180,E1 -19495.847,E2 -19495.847} C_VEL
LIN {X 0,Y 253.028,Z 560.407,A -85,B 0,C 180,E1 -19497.679,E2 -19497.679} C_VEL
LIN {X 0,Y 249.085,Z 572.255,A -85,B 0,C 180,E1 -19499.947,E2 -19499.947} C_VEL
LIN {X 0,Y 245.665,Z 582.234,A -85,B 0,C 180,E1 -19502.298,E2 -19502.298} C_VEL
LIN {X 0,Y 242.264,Z 592.004,A -85,B 0,C 180,E1 -19505.126,E2 -19505.126} C_VEL
LIN {X 0,Y 239.251,Z 600.157,A -85,B 0,C 180,E1 -19508.005,E2 -19508.005} C_VEL
LIN {X 0,Y 236.924,Z 606.909,A -85,B 0,C 180,E1 -19510.956,E2 -19510.956} C_VEL
LIN {X 0,Y 234.928,Z 613.148,A -85,B 0,C 180,E1 -19514.381,E2 -19514.381} C_VEL
LIN {X 0,Y 233.584,Z 617.979,A -85,B 0,C 180,E1 -19517.842,E2 -19517.842} C_VEL
LIN {X 0,Y 232.918,Z 621.527,A -85,B 0,C 180,E1 -19521.323,E2 -19521.323} C_VEL
LIN {X 0,Y 232.684,Z 623.864,A -85,B 0,C 180,E1 -19524.801,E2 -19524.801} C_VEL
LIN {X 0,Y 232.74,Z 625.042,A -85,B 0,C 180,E1 -19528.27,E2 -19528.27} C_VEL
LIN {X 0,Y 232.801,Z 625.197,A -85,B 0,C 180,E1 -19530,E2 -19530} C_VEL
LIN {X 0,Y 232.652,Z 624.582,A -85,B 0,C 180,E1 -19533.464,E2 -19533.464} C_VEL
LIN {X 0,Y 232.705,Z 622.811,A -85,B 0,C 180,E1 -19536.938,E2 -19536.938} C_VEL
LIN {X 0,Y 233.174,Z 619.866,A -85,B 0,C 180,E1 -19540.419,E2 -19540.419} C_VEL
LIN {X 0,Y 234.2,Z 615.679,A -85,B 0,C 180,E1 -19543.89,E2 -19543.89} C_VEL
LIN {X 0,Y 235.803,Z 609.854,A -85,B 0,C 180,E1 -19547.495,E2 -19547.495} C_VEL
LIN {X 0,Y 238.17,Z 603.106,A -85,B 0,C 180,E1 -19550.738,E2 -19550.738} C_VEL
LIN {X 0,Y 241.365,Z 594.365,A -85,B 0,C 180,E1 -19554.056,E2 -19554.056} C_VEL
LIN {X 0,Y 244.659,Z 585.021,A -85,B 0,C 180,E1 -19556.918,E2 -19556.918} C_VEL
LIN {X 0,Y 247.89,Z 575.652,A -85,B 0,C 180,E1 -19559.278,E2 -19559.278} C_VEL
LIN {X 0,Y 252.007,Z 563.427,A -85,B 0,C 180,E1 -19561.761,E2 -19561.761} C_VEL
LIN {X 0,Y 255.484,Z 552.193,A -85,B 0,C 180,E1 -19563.614,E2 -19563.614} C_VEL
LIN {X 0,Y 259.314,Z 538.256,A -85,B 0,C 180,E1 -19565.475,E2 -19565.475} C_VEL
LIN {X 0,Y 262.771,Z 523.625,A -85,B 0,C 180,E1 -19566.996,E2 -19566.996} C_VEL
LIN {X 0,Y 265.527,Z 509.834,A -85,B 0,C 180,E1 -19568.099,E2 -19568.099} C_VEL
LIN {X 0,Y 267.961,Z 494.394,A -85,B 0,C 180,E1 -19569.009,E2 -19569.009} C_VEL
LIN {X 0,Y 269.567,Z 479.11,A -85,B 0,C 180,E1 -19569.637,E2 -19569.637} C_VEL
LIN {X 0,Y 274.022,Z 395.693,A -85,B 0,C 180,E1 -19571.724,E2 -19571.724} C_VEL
LIN {X 0,Y 274.668,Z 381.378,A -85,B 0,C 180,E1 -19572.096,E2 -19572.096} C_VEL
LIN {X 0,Y 267.935,Z 365.691,A -85,B 0,C 180,E1 -19573.967,E2 -19573.967} C_VEL
LIN {X 0,Y 260.465,Z 350.814,A -85,B 0,C 180,E1 -19576.136,E2 -19576.136} C_VEL
LIN {X 0,Y 253.097,Z 337.68,A -85,B 0,C 180,E1 -19578.431,E2 -19578.431} C_VEL
LIN {X 0,Y 246.165,Z 326.69,A -85,B 0,C 180,E1 -19580.761,E2 -19580.761} C_VEL
LIN {X 0,Y 242.887,Z 321.707,A -85,B 0,C 180,E1 -19581.942,E2 -19581.942} C_VEL
LIN {X 0,Y 239.162,Z 316.298,A -85,B 0,C 180,E1 -19583.352,E2 -19583.352} C_VEL
LIN {X 0,Y 236.55,Z 312.664,A -85,B 0,C 180,E1 -19584.388,E2 -19584.388} C_VEL
LIN {X 0,Y 235.603,Z 311.145,A -85,B 0,C 180,E1 -19584.787,E2 -19584.787} C_VEL
LIN {X 0,Y 234.922,Z 308.843,A -85,B 0,C 180,E1 -19586.204,E2 -19586.204} C_VEL
LIN {X 0,Y 234.916,Z 308.841,A -85,B 0,C 180,E1 -19590.178,E2 -19590.178} C_VEL
LIN {X 0,Y 234.934,Z 308.842,A -85,B 0,C 180,E1 -19593.821,E2 -19593.821} C_VEL
LIN {X 0,Y 234.93,Z 308.83,A -85,B 0,C 180,E1 -19598.962,E2 -19598.962} C_VEL
LIN {X 0,Y 235.048,Z 308.812,A -85,B 0,C 180,E1 -19603.093,E2 -19603.093} C_VEL
LIN {X 0,Y 235.086,Z 308.784,A -85,B 0,C 180,E1 -19607.921,E2 -19607.921} C_VEL
LIN {X 0,Y 235.29,Z 308.795,A -85,B 0,C 180,E1 -19611.411,E2 -19611.411} C_VEL
LIN {X 0,Y 235.335,Z 308.792,A -85,B 0,C 180,E1 -19613.14,E2 -19613.14} C_VEL
LIN {X 0,Y 235.571,Z 308.755,A -85,B 0,C 180,E1 -19618.291,E2 -19618.291} C_VEL
LIN {X 0,Y 235.57,Z 308.76,A -85,B 0,C 180,E1 -19621.71,E2 -19621.71} C_VEL
LIN {X 0,Y 235.349,Z 308.783,A -85,B 0,C 180,E1 -19626.86,E2 -19626.86} C_VEL
LIN {X 0,Y 235.179,Z 308.807,A -85,B 0,C 180,E1 -19630.329,E2 -19630.329} C_VEL
LIN {X 0,Y 235.064,Z 308.822,A -85,B 0,C 180,E1 -19635.61,E2 -19635.61} C_VEL
LIN {X 0,Y 234.964,Z 308.811,A -85,B 0,C 180,E1 -19639.21,E2 -19639.21} C_VEL
LIN {X 0,Y 234.937,Z 308.83,A -85,B 0,C 180,E1 -19642.885,E2 -19642.885} C_VEL
LIN {X 0,Y 234.952,Z 308.813,A -85,B 0,C 180,E1 -19646.66,E2 -19646.66} C_VEL
LIN {X 0,Y 234.916,Z 308.849,A -85,B 0,C 180,E1 -19650.57,E2 -19650.57} C_VEL
LIN {X 0,Y 234.926,Z 308.84,A -85,B 0,C 180,E1 -19654.639,E2 -19654.639} C_VEL
LIN {X 0,Y 234.937,Z 308.863,A -85,B 0,C 180,E1 -19655.313,E2 -19655.313} C_VEL
LIN {X 0,Y 235.756,Z 311.341,A -85,B 0,C 180,E1 -19655.723,E2 -19655.723} C_VEL
LIN {X 0,Y 237.748,Z 313.643,A -85,B 0,C 180,E1 -19656.506,E2 -19656.506} C_VEL
LIN {X 0,Y 238.837,Z 314.526,A -85,B 0,C 180,E1 -19656.904,E2 -19656.904} C_VEL
LIN {X 0,Y 240.896,Z 317.849,A -85,B 0,C 180,E1 -19657.716,E2 -19657.716} C_VEL
LIN {X 0,Y 242.705,Z 319.8,A -85,B 0,C 180,E1 -19658.362,E2 -19658.362} C_VEL
LIN {X 0,Y 245.311,Z 323.404,A -85,B 0,C 180,E1 -19659.294,E2 -19659.294} C_VEL
LIN {X 0,Y 250.128,Z 330.066,A -85,B 0,C 180,E1 -19660.923,E2 -19660.923} C_VEL
LIN {X 0,Y 257.503,Z 340.787,A -85,B 0,C 180,E1 -19663.226,E2 -19663.226} C_VEL
LIN {X 0,Y 264.241,Z 351.503,A -85,B 0,C 180,E1 -19665.176,E2 -19665.176} C_VEL
LIN {X 0,Y 268.842,Z 360.075,A -85,B 0,C 180,E1 -19666.462,E2 -19666.462} C_VEL
LIN {X 0,Y 275.046,Z 373.558,A -85,B 0,C 180,E1 -19668.153,E2 -19668.153} C_VEL
LIN {X 0,Y 270.097,Z 467.53,A -85,B 0,C 180,E1 -19670.517,E2 -19670.517} C_VEL
LIN {X 0,Y 268.496,Z 482.674,A -85,B 0,C 180,E1 -19671.143,E2 -19671.143} C_VEL
LIN {X 0,Y 266.238,Z 498.561,A -85,B 0,C 180,E1 -19672.141,E2 -19672.141} C_VEL
LIN {X 0,Y 263.9,Z 511.041,A -85,B 0,C 180,E1 -19673.168,E2 -19673.168} C_VEL
LIN {X 0,Y 260.946,Z 524.756,A -85,B 0,C 180,E1 -19674.617,E2 -19674.617} C_VEL
LIN {X 0,Y 257.572,Z 537.226,A -85,B 0,C 180,E1 -19676.225,E2 -19676.225} C_VEL
LIN {X 0,Y 253.863,Z 549.854,A -85,B 0,C 180,E1 -19678.265,E2 -19678.265} C_VEL
LIN {X 0,Y 250.173,Z 560.888,A -85,B 0,C 180,E1 -19680.445,E2 -19680.445} C_VEL
LIN {X 0,Y 246.824,Z 570.932,A -85,B 0,C 180,E1 -19682.899,E2 -19682.899} C_VEL
LIN {X 0,Y 243.31,Z 580.373,A -85,B 0,C 180,E1 -19685.695,E2 -19685.695} C_VEL
LIN {X 0,Y 240.329,Z 588.227,A -85,B 0,C 180,E1 -19688.56,E2 -19688.56} C_VEL
LIN {X 0,Y 237.626,Z 595.552,A -85,B 0,C 180,E1 -19691.908,E2 -19691.908} C_VEL
LIN {X 0,Y 235.585,Z 601.359,A -85,B 0,C 180,E1 -19695.311,E2 -19695.311} C_VEL
LIN {X 0,Y 234.524,Z 604.794,A -85,B 0,C 180,E1 -19697.892,E2 -19697.892} C_VEL
LIN {X 0,Y 233.557,Z 608.268,A -85,B 0,C 180,E1 -19701.347,E2 -19701.347} C_VEL
LIN {X 0,Y 232.989,Z 610.562,A -85,B 0,C 180,E1 -19704.808,E2 -19704.808} C_VEL
LIN {X 0,Y 232.822,Z 611.728,A -85,B 0,C 180,E1 -19708.27,E2 -19708.27} C_VEL
LIN {X 0,Y 232.821,Z 611.741,A -85,B 0,C 180,E1 -19711.73,E2 -19711.73} C_VEL
LIN {X 0,Y 233.029,Z 610.449,A -85,B 0,C 180,E1 -19715.581,E2 -19715.581} C_VEL
LIN {X 0,Y 233.481,Z 608.381,A -85,B 0,C 180,E1 -19718.656,E2 -19718.656} C_VEL
LIN {X 0,Y 234.467,Z 604.951,A -85,B 0,C 180,E1 -19722.111,E2 -19722.111} C_VEL
LIN {X 0,Y 236.047,Z 600.249,A -85,B 0,C 180,E1 -19725.543,E2 -19725.543} C_VEL
LIN {X 0,Y 238.231,Z 594.153,A -85,B 0,C 180,E1 -19728.935,E2 -19728.935} C_VEL
LIN {X 0,Y 241.064,Z 586.473,A -85,B 0,C 180,E1 -19732.271,E2 -19732.271} C_VEL
LIN {X 0,Y 244.164,Z 578.279,A -85,B 0,C 180,E1 -19735.122,E2 -19735.122} C_VEL
LIN {X 0,Y 247.786,Z 568.402,A -85,B 0,C 180,E1 -19737.903,E2 -19737.903} C_VEL
LIN {X 0,Y 251.144,Z 558.278,A -85,B 0,C 180,E1 -19740.245,E2 -19740.245} C_VEL
LIN {X 0,Y 255.114,Z 546.208,A -85,B 0,C 180,E1 -19742.492,E2 -19742.492} C_VEL
LIN {X 0,Y 258.207,Z 535.39,A -85,B 0,C 180,E1 -19744.15,E2 -19744.15} C_VEL
LIN {X 0,Y 261.518,Z 522.521,A -85,B 0,C 180,E1 -19745.767,E2 -19745.767} C_VEL
LIN {X 0,Y 264.307,Z 509.515,A -85,B 0,C 180,E1 -19747.088,E2 -19747.088} C_VEL
LIN {X 0,Y 266.865,Z 494.997,A -85,B 0,C 180,E1 -19748.233,E2 -19748.233} C_VEL
LIN {X 0,Y 268.891,Z 480.221,A -85,B 0,C 180,E1 -19749.09,E2 -19749.09} C_VEL
LIN {X 0,Y 270.371,Z 465.081,A -85,B 0,C 180,E1 -19749.677,E2 -19749.677} C_VEL
LIN {X 0,Y 275.129,Z 374.348,A -85,B 0,C 180,E1 -19751.944,E2 -19751.944} C_VEL
LIN {X 0,Y 274.827,Z 372.83,A -85,B 0,C 180,E1 -19752.054,E2 -19752.054} C_VEL
LIN {X 0,Y 267.832,Z 357.914,A -85,B 0,C 180,E1 -19753.971,E2 -19753.971} C_VEL
LIN {X 0,Y 263.312,Z 349.836,A -85,B 0,C 180,E1 -19755.24,E2 -19755.24} C_VEL
LIN {X 0,Y 255.714,Z 338.067,A -85,B 0,C 180,E1 -19757.473,E2 -19757.473} C_VEL
LIN {X 0,Y 248.615,Z 327.794,A -85,B 0,C 180,E1 -19759.75,E2 -19759.75} C_VEL
LIN {X 0,Y 245.212,Z 323.289,A -85,B 0,C 180,E1 -19760.91,E2 -19760.91} C_VEL
LIN {X 0,Y 242.605,Z 319.598,A -85,B 0,C 180,E1 -19761.853,E2 -19761.853} C_VEL
LIN {X 0,Y 239.692,Z 316.17,A -85,B 0,C 180,E1 -19762.921,E2 -19762.921} C_VEL
LIN {X 0,Y 238.577,Z 314.167,A -85,B 0,C 180,E1 -19763.378,E2 -19763.378} C_VEL
LIN {X 0,Y 236.26,Z 312.151,A -85,B 0,C 180,E1 -19764.25,E2 -19764.25} C_VEL
LIN {X 0,Y 235.117,Z 309.751,A -85,B 0,C 180,E1 -19764.766,E2 -19764.766} C_VEL
LIN {X 0,Y 234.926,Z 308.829,A -85,B 0,C 180,E1 -19764.943,E2 -19764.943} C_VEL
LIN {X 0,Y 234.948,Z 308.824,A -85,B 0,C 180,E1 -19767.423,E2 -19767.423} C_VEL
LIN {X 0,Y 234.911,Z 308.831,A -85,B 0,C 180,E1 -19771.4,E2 -19771.4} C_VEL
LIN {X 0,Y 234.963,Z 308.835,A -85,B 0,C 180,E1 -19775.244,E2 -19775.244} C_VEL
LIN {X 0,Y 234.964,Z 308.833,A -85,B 0,C 180,E1 -19778.965,E2 -19778.965} C_VEL
LIN {X 0,Y 235.051,Z 308.822,A -85,B 0,C 180,E1 -19783.092,E2 -19783.092} C_VEL
LIN {X 0,Y 235.092,Z 308.822,A -85,B 0,C 180,E1 -19787.921,E2 -19787.921} C_VEL
LIN {X 0,Y 235.316,Z 308.786,A -85,B 0,C 180,E1 -19791.412,E2 -19791.412} C_VEL
LIN {X 0,Y 235.352,Z 308.795,A -85,B 0,C 180,E1 -19793.14,E2 -19793.14} C_VEL
LIN {X 0,Y 235.263,Z 308.795,A -85,B 0,C 180,E1 -19796.492,E2 -19796.492} C_VEL
LIN {X 0,Y 235.03,Z 308.834,A -85,B 0,C 180,E1 -19797.45,E2 -19797.45} C_VEL
LIN {X 0,Y 233.748,Z 308.996,A -85,B 0,C 180,E1 -19798.866,E2 -19798.866} C_VEL
LIN {X 0,Y 229.38,Z 309.538,A -85,B 0,C 180,E1 -19802.166,E2 -19802.166} C_VEL
LIN {X 0,Y 228.267,Z 309.669,A -85,B 0,C 180,E1 -19803.646,E2 -19803.646} C_VEL
LIN {X 0,Y 228.159,Z 309.678,A -85,B 0,C 180,E1 -19804.149,E2 -19804.149} C_VEL
LIN {X 0,Y 228.302,Z 309.673,A -85,B 0,C 180,E1 -19807.073,E2 -19807.073} C_VEL
LIN {X 0,Y 228.136,Z 309.69,A -85,B 0,C 180,E1 -19810.651,E2 -19810.651} C_VEL
LIN {X 0,Y 228.011,Z 309.711,A -85,B 0,C 180,E1 -19816.105,E2 -19816.105} C_VEL
LIN {X 0,Y 227.914,Z 309.712,A -85,B 0,C 180,E1 -19821.718,E2 -19821.718} C_VEL
LIN {X 0,Y 227.897,Z 309.715,A -85,B 0,C 180,E1 -19826.583,E2 -19826.583} C_VEL
LIN {X 0,Y 227.867,Z 309.725,A -85,B 0,C 180,E1 -19830.281,E2 -19830.281} C_VEL
LIN {X 0,Y 227.879,Z 309.808,A -85,B 0,C 180,E1 -19831.75,E2 -19831.75} C_VEL
LIN {X 0,Y 228.234,Z 311.112,A -85,B 0,C 180,E1 -19832.411,E2 -19832.411} C_VEL
LIN {X 0,Y 229.561,Z 313.474,A -85,B 0,C 180,E1 -19833.058,E2 -19833.058} C_VEL
LIN {X 0,Y 231.721,Z 315.984,A -85,B 0,C 180,E1 -19834,E2 -19834} C_VEL
LIN {X 0,Y 233.486,Z 318.244,A -85,B 0,C 180,E1 -19834.752,E2 -19834.752} C_VEL
LIN {X 0,Y 236.405,Z 322.354,A -85,B 0,C 180,E1 -19835.96,E2 -19835.96} C_VEL
LIN {X 0,Y 241.244,Z 329.648,A -85,B 0,C 180,E1 -19837.852,E2 -19837.852} C_VEL
LIN {X 0,Y 247.719,Z 340.018,A -85,B 0,C 180,E1 -19840.185,E2 -19840.185} C_VEL
LIN {X 0,Y 254.797,Z 352.403,A -85,B 0,C 180,E1 -19842.53,E2 -19842.53} C_VEL
LIN {X 0,Y 261.356,Z 365.366,A -85,B 0,C 180,E1 -19844.563,E2 -19844.563} C_VEL
LIN {X 0,Y 268.008,Z 380.181,A -85,B 0,C 180,E1 -19846.517,E2 -19846.517} C_VEL
LIN {X 0,Y 269.41,Z 383.657,A -85,B 0,C 180,E1 -19846.922,E2 -19846.922} C_VEL
LIN {X 0,Y 264.742,Z 472.649,A -85,B 0,C 180,E1 -19849.179,E2 -19849.179} C_VEL
LIN {X 0,Y 263.424,Z 487.601,A -85,B 0,C 180,E1 -19849.687,E2 -19849.687} C_VEL
LIN {X 0,Y 261.373,Z 502.371,A -85,B 0,C 180,E1 -19850.438,E2 -19850.438} C_VEL
LIN {X 0,Y 258.641,Z 516.846,A -85,B 0,C 180,E1 -19851.446,E2 -19851.446} C_VEL
LIN {X 0,Y 255.458,Z 530.922,A -85,B 0,C 180,E1 -19852.754,E2 -19852.754} C_VEL
LIN {X 0,Y 251.918,Z 544.505,A -85,B 0,C 180,E1 -19854.384,E2 -19854.384} C_VEL
LIN {X 0,Y 247.728,Z 558.059,A -85,B 0,C 180,E1 -19856.413,E2 -19856.413} C_VEL
LIN {X 0,Y 243.583,Z 570.263,A -85,B 0,C 180,E1 -19858.713,E2 -19858.713} C_VEL
LIN {X 0,Y 239.898,Z 580.516,A -85,B 0,C 180,E1 -19861.095,E2 -19861.095} C_VEL
LIN {X 0,Y 236.738,Z 589.182,A -85,B 0,C 180,E1 -19863.558,E2 -19863.558} C_VEL
LIN {X 0,Y 233.428,Z 597.746,A -85,B 0,C 180,E1 -19866.49,E2 -19866.49} C_VEL
LIN {X 0,Y 230.759,Z 604.879,A -85,B 0,C 180,E1 -19869.498,E2 -19869.498} C_VEL
LIN {X 0,Y 228.507,Z 611.506,A -85,B 0,C 180,E1 -19873.012,E2 -19873.012} C_VEL
LIN {X 0,Y 226.911,Z 616.696,A -85,B 0,C 180,E1 -19876.568,E2 -19876.568} C_VEL
LIN {X 0,Y 226.144,Z 619.704,A -85,B 0,C 180,E1 -19879.254,E2 -19879.254} C_VEL
LIN {X 0,Y 225.67,Z 622.639,A -85,B 0,C 180,E1 -19882.844,E2 -19882.844} C_VEL
LIN {X 0,Y 225.549,Z 624.391,A -85,B 0,C 180,E1 -19886.427,E2 -19886.427} C_VEL
LIN {X 0,Y 225.714,Z 624.995,A -85,B 0,C 180,E1 -19890,E2 -19890} C_VEL
LIN {X 0,Y 225.548,Z 624.378,A -85,B 0,C 180,E1 -19893.573,E2 -19893.573} C_VEL
LIN {X 0,Y 225.617,Z 622.607,A -85,B 0,C 180,E1 -19897.157,E2 -19897.157} C_VEL
LIN {X 0,Y 226.138,Z 619.66,A -85,B 0,C 180,E1 -19900.747,E2 -19900.747} C_VEL
LIN {X 0,Y 227.253,Z 615.473,A -85,B 0,C 180,E1 -19904.324,E2 -19904.324} C_VEL
LIN {X 0,Y 228.884,Z 609.931,A -85,B 0,C 180,E1 -19907.881,E2 -19907.881} C_VEL
LIN {X 0,Y 231.462,Z 602.899,A -85,B 0,C 180,E1 -19911.368,E2 -19911.368} C_VEL
LIN {X 0,Y 234.352,Z 595.383,A -85,B 0,C 180,E1 -19914.352,E2 -19914.352} C_VEL
LIN {X 0,Y 237.589,Z 586.705,A -85,B 0,C 180,E1 -19917.157,E2 -19917.157} C_VEL
LIN {X 0,Y 241.054,Z 577.085,A -85,B 0,C 180,E1 -19919.711,E2 -19919.711} C_VEL
LIN {X 0,Y 244.936,Z 566.209,A -85,B 0,C 180,E1 -19922.06,E2 -19922.06} C_VEL
LIN {X 0,Y 248.796,Z 554.339,A -85,B 0,C 180,E1 -19924.154,E2 -19924.154} C_VEL
LIN {X 0,Y 252.778,Z 540.913,A -85,B 0,C 180,E1 -19926.045,E2 -19926.045} C_VEL
LIN {X 0,Y 256.267,Z 527.022,A -85,B 0,C 180,E1 -19927.602,E2 -19927.602} C_VEL
LIN {X 0,Y 259.263,Z 513.018,A -85,B 0,C 180,E1 -19928.818,E2 -19928.818} C_VEL
LIN {X 0,Y 261.886,Z 498.03,A -85,B 0,C 180,E1 -19929.781,E2 -19929.781} C_VEL
LIN {X 0,Y 263.819,Z 482.349,A -85,B 0,C 180,E1 -19930.49,E2 -19930.49} C_VEL
LIN {X 0,Y 265.223,Z 462.475,A -85,B 0,C 180,E1 -19931.045,E2 -19931.045} C_VEL
LIN {X 0,Y 269.298,Z 383.499,A -85,B 0,C 180,E1 -19933.053,E2 -19933.053} C_VEL
LIN {X 0,Y 263.07,Z 369.051,A -85,B 0,C 180,E1 -19934.864,E2 -19934.864} C_VEL
LIN {X 0,Y 256.102,Z 355.01,A -85,B 0,C 180,E1 -19936.985,E2 -19936.985} C_VEL
LIN {X 0,Y 249.338,Z 342.744,A -85,B 0,C 180,E1 -19939.188,E2 -19939.188} C_VEL
LIN {X 0,Y 242.667,Z 331.944,A -85,B 0,C 180,E1 -19941.531,E2 -19941.531} C_VEL
LIN {X 0,Y 239.675,Z 327.315,A -85,B 0,C 180,E1 -19942.655,E2 -19942.655} C_VEL
LIN {X 0,Y 236.054,Z 321.96,A -85,B 0,C 180,E1 -19944.082,E2 -19944.082} C_VEL
LIN {X 0,Y 233.322,Z 317.977,A -85,B 0,C 180,E1 -19945.22,E2 -19945.22} C_VEL
LIN {X 0,Y 229.811,Z 313.759,A -85,B 0,C 180,E1 -19946.724,E2 -19946.724} C_VEL
LIN {X 0,Y 228.257,Z 311.224,A -85,B 0,C 180,E1 -19947.462,E2 -19947.462} C_VEL
LIN {X 0,Y 228.078,Z 310.632,A -85,B 0,C 180,E1 -19947.63,E2 -19947.63} C_VEL
LIN {X 0,Y 227.861,Z 309.724,A -85,B 0,C 180,E1 -19948.247,E2 -19948.247} C_VEL
LIN {X 0,Y 227.837,Z 309.723,A -85,B 0,C 180,E1 -19952.439,E2 -19952.439} C_VEL
LIN {X 0,Y 227.849,Z 309.722,A -85,B 0,C 180,E1 -19956.36,E2 -19956.36} C_VEL
LIN {X 0,Y 227.883,Z 309.69,A -85,B 0,C 180,E1 -19960.169,E2 -19960.169} C_VEL
LIN {X 0,Y 228.011,Z 309.703,A -85,B 0,C 180,E1 -19963.895,E2 -19963.895} C_VEL
LIN {X 0,Y 228.044,Z 309.663,A -85,B 0,C 180,E1 -19967.542,E2 -19967.542} C_VEL
LIN {X 0,Y 228.232,Z 309.666,A -85,B 0,C 180,E1 -19971.143,E2 -19971.143} C_VEL
LIN {X 0,Y 228.287,Z 309.672,A -85,B 0,C 180,E1 -19972.927,E2 -19972.927} C_VEL
LIN {X 0,Y 228.529,Z 309.633,A -85,B 0,C 180,E1 -19978.238,E2 -19978.238} C_VEL
LIN {X 0,Y 228.529,Z 309.636,A -85,B 0,C 180,E1 -19981.763,E2 -19981.763} C_VEL
LIN {X 0,Y 228.301,Z 309.661,A -85,B 0,C 180,E1 -19987.073,E2 -19987.073} C_VEL
LIN {X 0,Y 228.121,Z 309.685,A -85,B 0,C 180,E1 -19990.653,E2 -19990.653} C_VEL
LIN {X 0,Y 228.011,Z 309.704,A -85,B 0,C 180,E1 -19996.106,E2 -19996.106} C_VEL
LIN {X 0,Y 227.913,Z 309.686,A -85,B 0,C 180,E1 -20001.718,E2 -20001.718} C_VEL
LIN {X 0,Y 227.928,Z 309.688,A -85,B 0,C 180,E1 -20006.598,E2 -20006.598} C_VEL
LIN {X 0,Y 227.89,Z 309.723,A -85,B 0,C 180,E1 -20010.291,E2 -20010.291} C_VEL
LIN {X 0,Y 227.9,Z 309.724,A -85,B 0,C 180,E1 -20012.76,E2 -20012.76} C_VEL
LIN {X 0,Y 228.669,Z 312.184,A -85,B 0,C 180,E1 -20013.2,E2 -20013.2} C_VEL
LIN {X 0,Y 230.598,Z 314.48,A -85,B 0,C 180,E1 -20014.057,E2 -20014.057} C_VEL
LIN {X 0,Y 231.976,Z 315.472,A -85,B 0,C 180,E1 -20014.615,E2 -20014.615} C_VEL
LIN {X 0,Y 233.952,Z 318.706,A -85,B 0,C 180,E1 -20015.485,E2 -20015.485} C_VEL
LIN {X 0,Y 235.975,Z 320.781,A -85,B 0,C 180,E1 -20016.279,E2 -20016.279} C_VEL
LIN {X 0,Y 238.512,Z 324.312,A -85,B 0,C 180,E1 -20017.281,E2 -20017.281} C_VEL
LIN {X 0,Y 239.931,Z 326.143,A -85,B 0,C 180,E1 -20017.815,E2 -20017.815} C_VEL
LIN {X 0,Y 246.273,Z 334.839,A -85,B 0,C 180,E1 -20020.082,E2 -20020.082} C_VEL
LIN {X 0,Y 253.983,Z 346.311,A -85,B 0,C 180,E1 -20022.596,E2 -20022.596} C_VEL
LIN {X 0,Y 260.48,Z 356.842,A -85,B 0,C 180,E1 -20024.548,E2 -20024.548} C_VEL
LIN {X 0,Y 265.071,Z 365.691,A -85,B 0,C 180,E1 -20025.885,E2 -20025.885} C_VEL
LIN {X 0,Y 269.682,Z 375.835,A -85,B 0,C 180,E1 -20027.197,E2 -20027.197} C_VEL
LIN {X 0,Y 264.675,Z 467.748,A -85,B 0,C 180,E1 -20029.543,E2 -20029.543} C_VEL
LIN {X 0,Y 263.018,Z 482.888,A -85,B 0,C 180,E1 -20030.175,E2 -20030.175} C_VEL
LIN {X 0,Y 260.855,Z 497.612,A -85,B 0,C 180,E1 -20031.092,E2 -20031.092} C_VEL
LIN {X 0,Y 258.106,Z 512.005,A -85,B 0,C 180,E1 -20032.292,E2 -20032.292} C_VEL
LIN {X 0,Y 254.815,Z 526.515,A -85,B 0,C 180,E1 -20033.877,E2 -20033.877} C_VEL
LIN {X 0,Y 251.341,Z 538.72,A -85,B 0,C 180,E1 -20035.513,E2 -20035.513} C_VEL
LIN {X 0,Y 247.488,Z 551.125,A -85,B 0,C 180,E1 -20037.589,E2 -20037.589} C_VEL
LIN {X 0,Y 243.317,Z 563.065,A -85,B 0,C 180,E1 -20040.058,E2 -20040.058} C_VEL
LIN {X 0,Y 239.916,Z 572.616,A -85,B 0,C 180,E1 -20042.525,E2 -20042.525} C_VEL
LIN {X 0,Y 236.355,Z 581.8,A -85,B 0,C 180,E1 -20045.4,E2 -20045.4} C_VEL
LIN {X 0,Y 233.297,Z 589.432,A -85,B 0,C 180,E1 -20048.345,E2 -20048.345} C_VEL
LIN {X 0,Y 230.842,Z 595.758,A -85,B 0,C 180,E1 -20051.357,E2 -20051.357} C_VEL
LIN {X 0,Y 228.714,Z 601.564,A -85,B 0,C 180,E1 -20054.86,E2 -20054.86} C_VEL
LIN {X 0,Y 227.54,Z 604.999,A -85,B 0,C 180,E1 -20057.514,E2 -20057.514} C_VEL
LIN {X 0,Y 226.521,Z 608.472,A -85,B 0,C 180,E1 -20061.076,E2 -20061.076} C_VEL
LIN {X 0,Y 225.923,Z 610.765,A -85,B 0,C 180,E1 -20064.645,E2 -20064.645} C_VEL
LIN {X 0,Y 225.739,Z 611.931,A -85,B 0,C 180,E1 -20068.216,E2 -20068.216} C_VEL
LIN {X 0,Y 225.738,Z 611.943,A -85,B 0,C 180,E1 -20071.784,E2 -20071.784} C_VEL
LIN {X 0,Y 225.918,Z 610.787,A -85,B 0,C 180,E1 -20075.449,E2 -20075.449} C_VEL
LIN {X 0,Y 226.462,Z 608.584,A -85,B 0,C 180,E1 -20078.926,E2 -20078.926} C_VEL
LIN {X 0,Y 227.492,Z 605.154,A -85,B 0,C 180,E1 -20082.489,E2 -20082.489} C_VEL
LIN {X 0,Y 229.198,Z 600.451,A -85,B 0,C 180,E1 -20086.019,E2 -20086.019} C_VEL
LIN {X 0,Y 231.499,Z 594.356,A -85,B 0,C 180,E1 -20089.508,E2 -20089.508} C_VEL
LIN {X 0,Y 234.473,Z 586.675,A -85,B 0,C 180,E1 -20092.932,E2 -20092.932} C_VEL
LIN {X 0,Y 237.717,Z 578.481,A -85,B 0,C 180,E1 -20095.853,E2 -20095.853} C_VEL
LIN {X 0,Y 241.5,Z 568.604,A -85,B 0,C 180,E1 -20098.696,E2 -20098.696} C_VEL
LIN {X 0,Y 245.036,Z 558.478,A -85,B 0,C 180,E1 -20101.081,E2 -20101.081} C_VEL
LIN {X 0,Y 249.148,Z 546.408,A -85,B 0,C 180,E1 -20103.37,E2 -20103.37} C_VEL
LIN {X 0,Y 252.368,Z 535.589,A -85,B 0,C 180,E1 -20105.054,E2 -20105.054} C_VEL
LIN {X 0,Y 255.78,Z 522.719,A -85,B 0,C 180,E1 -20106.698,E2 -20106.698} C_VEL
LIN {X 0,Y 258.857,Z 508.953,A -85,B 0,C 180,E1 -20108.1,E2 -20108.1} C_VEL
LIN {X 0,Y 261.341,Z 495.191,A -85,B 0,C 180,E1 -20109.194,E2 -20109.194} C_VEL
LIN {X 0,Y 263.432,Z 480.412,A -85,B 0,C 180,E1 -20110.061,E2 -20110.061} C_VEL
LIN {X 0,Y 264.944,Z 465.264,A -85,B 0,C 180,E1 -20110.657,E2 -20110.657} C_VEL
LIN {X 0,Y 269.787,Z 376.69,A -85,B 0,C 180,E1 -20112.895,E2 -20112.895} C_VEL
LIN {X 0,Y 269.46,Z 375.189,A -85,B 0,C 180,E1 -20113.014,E2 -20113.014} C_VEL
LIN {X 0,Y 263.283,Z 361.881,A -85,B 0,C 180,E1 -20114.789,E2 -20114.789} C_VEL
LIN {X 0,Y 258.405,Z 353.252,A -85,B 0,C 180,E1 -20116.22,E2 -20116.22} C_VEL
LIN {X 0,Y 250.43,Z 340.858,A -85,B 0,C 180,E1 -20118.698,E2 -20118.698} C_VEL
LIN {X 0,Y 244.688,Z 332.628,A -85,B 0,C 180,E1 -20120.635,E2 -20120.635} C_VEL
LIN {X 0,Y 241.878,Z 328.782,A -85,B 0,C 180,E1 -20121.64,E2 -20121.64} C_VEL
LIN {X 0,Y 238.74,Z 324.549,A -85,B 0,C 180,E1 -20122.814,E2 -20122.814} C_VEL
LIN {X 0,Y 236.119,Z 320.997,A -85,B 0,C 180,E1 -20123.846,E2 -20123.846} C_VEL
LIN {X 0,Y 232.795,Z 317.107,A -85,B 0,C 180,E1 -20125.196,E2 -20125.196} C_VEL
LIN {X 0,Y 231.633,Z 315.108,A -85,B 0,C 180,E1 -20125.722,E2 -20125.722} C_VEL
LIN {X 0,Y 229.4,Z 313.264,A -85,B 0,C 180,E1 -20126.658,E2 -20126.658} C_VEL
LIN {X 0,Y 228.19,Z 311.019,A -85,B 0,C 180,E1 -20127.254,E2 -20127.254} C_VEL
LIN {X 0,Y 227.908,Z 309.699,A -85,B 0,C 180,E1 -20127.471,E2 -20127.471} C_VEL
LIN {X 0,Y 227.878,Z 309.693,A -85,B 0,C 180,E1 -20130.432,E2 -20130.432} C_VEL
LIN {X 0,Y 227.91,Z 309.711,A -85,B 0,C 180,E1 -20134.423,E2 -20134.423} C_VEL
LIN {X 0,Y 227.933,Z 309.707,A -85,B 0,C 180,E1 -20138.284,E2 -20138.284} C_VEL
LIN {X 0,Y 228.017,Z 309.706,A -85,B 0,C 180,E1 -20143.895,E2 -20143.895} C_VEL
LIN {X 0,Y 228.049,Z 309.695,A -85,B 0,C 180,E1 -20147.542,E2 -20147.542} C_VEL
LIN {X 0,Y 228.254,Z 309.665,A -85,B 0,C 180,E1 -20151.144,E2 -20151.144} C_VEL
LIN {X 0,Y 228.305,Z 309.671,A -85,B 0,C 180,E1 -20152.927,E2 -20152.927} C_VEL
LIN {X 0,Y 228.534,Z 309.643,A -85,B 0,C 180,E1 -20158.238,E2 -20158.238} C_VEL
LIN {X 0,Y 228.53,Z 309.641,A -85,B 0,C 180,E1 -20161.762,E2 -20161.762} C_VEL
LIN {X 0,Y 228.159,Z 309.678,A -85,B 0,C 180,E1 -20164.149,E2 -20164.149} C_VEL
LIN {X 0,Y 227.442,Z 309.773,A -85,B 0,C 180,E1 -20165.624,E2 -20165.624} C_VEL
LIN {X 0,Y 224.567,Z 310.131,A -85,B 0,C 180,E1 -20168.032,E2 -20168.032} C_VEL
LIN {X 0,Y 222.138,Z 310.436,A -85,B 0,C 180,E1 -20169.996,E2 -20169.996} C_VEL
LIN {X 0,Y 221.081,Z 310.574,A -85,B 0,C 180,E1 -20171.521,E2 -20171.521} C_VEL
LIN {X 0,Y 220.985,Z 310.575,A -85,B 0,C 180,E1 -20172.038,E2 -20172.038} C_VEL
LIN {X 0,Y 220.97,Z 310.582,A -85,B 0,C 180,E1 -20176.633,E2 -20176.633} C_VEL
LIN {X 0,Y 220.844,Z 310.601,A -85,B 0,C 180,E1 -20180.491,E2 -20180.491} C_VEL
LIN {X 0,Y 220.797,Z 310.607,A -85,B 0,C 180,E1 -20184.443,E2 -20184.443} C_VEL
LIN {X 0,Y 220.793,Z 310.607,A -85,B 0,C 180,E1 -20188.519,E2 -20188.519} C_VEL
LIN {X 0,Y 220.818,Z 310.612,A -85,B 0,C 180,E1 -20189.232,E2 -20189.232} C_VEL
LIN {X 0,Y 221.545,Z 312.958,A -85,B 0,C 180,E1 -20189.714,E2 -20189.714} C_VEL
LIN {X 0,Y 223.514,Z 315.345,A -85,B 0,C 180,E1 -20190.727,E2 -20190.727} C_VEL
LIN {X 0,Y 225.21,Z 316.581,A -85,B 0,C 180,E1 -20191.514,E2 -20191.514} C_VEL
LIN {X 0,Y 227.162,Z 319.753,A -85,B 0,C 180,E1 -20192.485,E2 -20192.485} C_VEL
LIN {X 0,Y 230.379,Z 323.719,A -85,B 0,C 180,E1 -20193.929,E2 -20193.929} C_VEL
LIN {X 0,Y 234.607,Z 330.04,A -85,B 0,C 180,E1 -20195.749,E2 -20195.749} C_VEL
LIN {X 0,Y 238.222,Z 335.527,A -85,B 0,C 180,E1 -20197.2,E2 -20197.2} C_VEL
LIN {X 0,Y 245.362,Z 347.289,A -85,B 0,C 180,E1 -20199.858,E2 -20199.858} C_VEL
LIN {X 0,Y 252.044,Z 359.513,A -85,B 0,C 180,E1 -20202.143,E2 -20202.143} C_VEL
LIN {X 0,Y 258.41,Z 372.547,A -85,B 0,C 180,E1 -20204.181,E2 -20204.181} C_VEL
LIN {X 0,Y 264.178,Z 386.018,A -85,B 0,C 180,E1 -20205.945,E2 -20205.945} C_VEL
LIN {X 0,Y 258.968,Z 478.466,A -85,B 0,C 180,E1 -20208.327,E2 -20208.327} C_VEL
LIN {X 0,Y 257.203,Z 493.813,A -85,B 0,C 180,E1 -20208.957,E2 -20208.957} C_VEL
LIN {X 0,Y 254.71,Z 508.685,A -85,B 0,C 180,E1 -20209.838,E2 -20209.838} C_VEL
LIN {X 0,Y 251.574,Z 523.624,A -85,B 0,C 180,E1 -20211.057,E2 -20211.057} C_VEL
LIN {X 0,Y 247.966,Z 537.662,A -85,B 0,C 180,E1 -20212.551,E2 -20212.551} C_VEL
LIN {X 0,Y 244.173,Z 550.805,A -85,B 0,C 180,E1 -20214.35,E2 -20214.35} C_VEL
LIN {X 0,Y 239.971,Z 563.224,A -85,B 0,C 180,E1 -20216.442,E2 -20216.442} C_VEL
LIN {X 0,Y 235.505,Z 575.407,A -85,B 0,C 180,E1 -20219.018,E2 -20219.018} C_VEL
LIN {X 0,Y 231.301,Z 586.326,A -85,B 0,C 180,E1 -20221.931,E2 -20221.931} C_VEL
LIN {X 0,Y 227.854,Z 595.294,A -85,B 0,C 180,E1 -20224.906,E2 -20224.906} C_VEL
LIN {X 0,Y 224.795,Z 602.798,A -85,B 0,C 180,E1 -20227.966,E2 -20227.966} C_VEL
LIN {X 0,Y 222.082,Z 610.043,A -85,B 0,C 180,E1 -20231.691,E2 -20231.691} C_VEL
LIN {X 0,Y 220.332,Z 615.324,A -85,B 0,C 180,E1 -20235.216,E2 -20235.216} C_VEL
LIN {X 0,Y 219.125,Z 619.5,A -85,B 0,C 180,E1 -20238.905,E2 -20238.905} C_VEL
LIN {X 0,Y 218.596,Z 622.435,A -85,B 0,C 180,E1 -20242.611,E2 -20242.611} C_VEL
LIN {X 0,Y 218.449,Z 624.188,A -85,B 0,C 180,E1 -20246.311,E2 -20246.311} C_VEL
LIN {X 0,Y 218.628,Z 624.792,A -85,B 0,C 180,E1 -20250,E2 -20250} C_VEL
LIN {X 0,Y 218.449,Z 624.174,A -85,B 0,C 180,E1 -20253.689,E2 -20253.689} C_VEL
LIN {X 0,Y 218.552,Z 622.403,A -85,B 0,C 180,E1 -20257.39,E2 -20257.39} C_VEL
LIN {X 0,Y 219.12,Z 619.455,A -85,B 0,C 180,E1 -20261.095,E2 -20261.095} C_VEL
LIN {X 0,Y 220.32,Z 615.268,A -85,B 0,C 180,E1 -20264.785,E2 -20264.785} C_VEL
LIN {X 0,Y 222.095,Z 609.726,A -85,B 0,C 180,E1 -20268.447,E2 -20268.447} C_VEL
LIN {X 0,Y 224.813,Z 602.692,A -85,B 0,C 180,E1 -20272.032,E2 -20272.032} C_VEL
LIN {X 0,Y 227.867,Z 595.177,A -85,B 0,C 180,E1 -20275.092,E2 -20275.092} C_VEL
LIN {X 0,Y 231.487,Z 585.885,A -85,B 0,C 180,E1 -20278.155,E2 -20278.155} C_VEL
LIN {X 0,Y 235.498,Z 575.237,A -85,B 0,C 180,E1 -20280.983,E2 -20280.983} C_VEL
LIN {X 0,Y 239.947,Z 563.011,A -85,B 0,C 180,E1 -20283.561,E2 -20283.561} C_VEL
LIN {X 0,Y 243.754,Z 551.779,A -85,B 0,C 180,E1 -20285.467,E2 -20285.467} C_VEL
LIN {X 0,Y 247.527,Z 538.822,A -85,B 0,C 180,E1 -20287.269,E2 -20287.269} C_VEL
LIN {X 0,Y 251.092,Z 525.043,A -85,B 0,C 180,E1 -20288.774,E2 -20288.774} C_VEL
LIN {X 0,Y 254.011,Z 511.679,A -85,B 0,C 180,E1 -20289.906,E2 -20289.906} C_VEL
LIN {X 0,Y 256.565,Z 497.054,A -85,B 0,C 180,E1 -20290.842,E2 -20290.842} C_VEL
LIN {X 0,Y 258.453,Z 482.132,A -85,B 0,C 180,E1 -20291.514,E2 -20291.514} C_VEL
LIN {X 0,Y 259.898,Z 462.25,A -85,B 0,C 180,E1 -20292.075,E2 -20292.075} C_VEL
LIN {X 0,Y 264.063,Z 385.904,A -85,B 0,C 180,E1 -20294.026,E2 -20294.026} C_VEL
LIN {X 0,Y 257.788,Z 371.252,A -85,B 0,C 180,E1 -20295.949,E2 -20295.949} C_VEL
LIN {X 0,Y 250.404,Z 356.395,A -85,B 0,C 180,E1 -20298.331,E2 -20298.331} C_VEL
LIN {X 0,Y 242.986,Z 343.268,A -85,B 0,C 180,E1 -20300.916,E2 -20300.916} C_VEL
LIN {X 0,Y 236.454,Z 332.809,A -85,B 0,C 180,E1 -20303.408,E2 -20303.408} C_VEL
LIN {X 0,Y 232.87,Z 327.471,A -85,B 0,C 180,E1 -20304.88,E2 -20304.88} C_VEL
LIN {X 0,Y 229.286,Z 322.291,A -85,B 0,C 180,E1 -20306.449,E2 -20306.449} C_VEL
LIN {X 0,Y 225.804,Z 317.812,A -85,B 0,C 180,E1 -20308.055,E2 -20308.055} C_VEL
LIN {X 0,Y 224.817,Z 316.147,A -85,B 0,C 180,E1 -20308.556,E2 -20308.556} C_VEL
LIN {X 0,Y 222.407,Z 314.259,A -85,B 0,C 180,E1 -20309.695,E2 -20309.695} C_VEL
LIN {X 0,Y 221.115,Z 311.879,A -85,B 0,C 180,E1 -20310.419,E2 -20310.419} C_VEL
LIN {X 0,Y 220.827,Z 310.598,A -85,B 0,C 180,E1 -20310.704,E2 -20310.704} C_VEL
LIN {X 0,Y 220.849,Z 310.594,A -85,B 0,C 180,E1 -20313.544,E2 -20313.544} C_VEL
LIN {X 0,Y 220.848,Z 310.601,A -85,B 0,C 180,E1 -20317.55,E2 -20317.55} C_VEL
LIN {X 0,Y 220.913,Z 310.563,A -85,B 0,C 180,E1 -20322.626,E2 -20322.626} C_VEL
LIN {X 0,Y 220.983,Z 310.546,A -85,B 0,C 180,E1 -20327.137,E2 -20327.137} C_VEL
LIN {X 0,Y 221.175,Z 310.538,A -85,B 0,C 180,E1 -20330.858,E2 -20330.858} C_VEL
LIN {X 0,Y 221.102,Z 310.557,A -85,B 0,C 180,E1 -20334.528,E2 -20334.528} C_VEL
LIN {X 0,Y 221.462,Z 310.513,A -85,B 0,C 180,E1 -20338.182,E2 -20338.182} C_VEL
LIN {X 0,Y 221.463,Z 310.516,A -85,B 0,C 180,E1 -20341.819,E2 -20341.819} C_VEL
LIN {X 0,Y 221.238,Z 310.542,A -85,B 0,C 180,E1 -20347.3,E2 -20347.3} C_VEL
LIN {X 0,Y 221.047,Z 310.565,A -85,B 0,C 180,E1 -20350.998,E2 -20350.998} C_VEL
LIN {X 0,Y 220.97,Z 310.585,A -85,B 0,C 180,E1 -20356.634,E2 -20356.634} C_VEL
LIN {X 0,Y 220.846,Z 310.56,A -85,B 0,C 180,E1 -20360.491,E2 -20360.491} C_VEL
LIN {X 0,Y 220.849,Z 310.6,A -85,B 0,C 180,E1 -20364.437,E2 -20364.437} C_VEL
LIN {X 0,Y 220.817,Z 310.575,A -85,B 0,C 180,E1 -20368.516,E2 -20368.516} C_VEL
LIN {X 0,Y 220.862,Z 310.588,A -85,B 0,C 180,E1 -20369.815,E2 -20369.815} C_VEL
LIN {X 0,Y 221.662,Z 313.113,A -85,B 0,C 180,E1 -20370.352,E2 -20370.352} C_VEL
LIN {X 0,Y 223.445,Z 315.283,A -85,B 0,C 180,E1 -20371.264,E2 -20371.264} C_VEL
LIN {X 0,Y 225.154,Z 316.47,A -85,B 0,C 180,E1 -20372.049,E2 -20372.049} C_VEL
LIN {X 0,Y 227.127,Z 319.752,A -85,B 0,C 180,E1 -20373.03,E2 -20373.03} C_VEL
LIN {X 0,Y 229.374,Z 321.95,A -85,B 0,C 180,E1 -20374.013,E2 -20374.013} C_VEL
LIN {X 0,Y 231.963,Z 325.518,A -85,B 0,C 180,E1 -20375.146,E2 -20375.146} C_VEL
LIN {X 0,Y 233.21,Z 326.952,A -85,B 0,C 180,E1 -20375.657,E2 -20375.657} C_VEL
LIN {X 0,Y 236.122,Z 330.781,A -85,B 0,C 180,E1 -20376.83,E2 -20376.83} C_VEL
LIN {X 0,Y 243.195,Z 340.779,A -85,B 0,C 180,E1 -20379.477,E2 -20379.477} C_VEL
LIN {X 0,Y 250.364,Z 351.601,A -85,B 0,C 180,E1 -20381.904,E2 -20381.904} C_VEL
LIN {X 0,Y 257.592,Z 363.611,A -85,B 0,C 180,E1 -20384.154,E2 -20384.154} C_VEL
LIN {X 0,Y 263.606,Z 376.436,A -85,B 0,C 180,E1 -20385.974,E2 -20385.974} C_VEL
LIN {X 0,Y 264.405,Z 378.178,A -85,B 0,C 180,E1 -20386.207,E2 -20386.207} C_VEL
LIN {X 0,Y 259.332,Z 467.966,A -85,B 0,C 180,E1 -20388.529,E2 -20388.529} C_VEL
LIN {X 0,Y 257.628,Z 483.101,A -85,B 0,C 180,E1 -20389.168,E2 -20389.168} C_VEL
LIN {X 0,Y 255.384,Z 497.823,A -85,B 0,C 180,E1 -20390.094,E2 -20390.094} C_VEL
LIN {X 0,Y 252.38,Z 512.897,A -85,B 0,C 180,E1 -20391.374,E2 -20391.374} C_VEL
LIN {X 0,Y 249.124,Z 526.722,A -85,B 0,C 180,E1 -20392.916,E2 -20392.916} C_VEL
LIN {X 0,Y 245.513,Z 538.927,A -85,B 0,C 180,E1 -20394.574,E2 -20394.574} C_VEL
LIN {X 0,Y 241.533,Z 551.331,A -85,B 0,C 180,E1 -20396.688,E2 -20396.688} C_VEL
LIN {X 0,Y 237.596,Z 562.074,A -85,B 0,C 180,E1 -20398.926,E2 -20398.926} C_VEL
LIN {X 0,Y 234.245,Z 571.344,A -85,B 0,C 180,E1 -20401.313,E2 -20401.313} C_VEL
LIN {X 0,Y 230.376,Z 580.785,A -85,B 0,C 180,E1 -20404.233,E2 -20404.233} C_VEL
LIN {X 0,Y 227.099,Z 588.638,A -85,B 0,C 180,E1 -20407.243,E2 -20407.243} C_VEL
LIN {X 0,Y 224.089,Z 595.964,A -85,B 0,C 180,E1 -20410.774,E2 -20410.774} C_VEL
LIN {X 0,Y 221.83,Z 601.769,A -85,B 0,C 180,E1 -20414.378,E2 -20414.378} C_VEL
LIN {X 0,Y 220.578,Z 605.204,A -85,B 0,C 180,E1 -20417.113,E2 -20417.113} C_VEL
LIN {X 0,Y 219.507,Z 608.676,A -85,B 0,C 180,E1 -20420.788,E2 -20420.788} C_VEL
LIN {X 0,Y 218.838,Z 611.026,A -85,B 0,C 180,E1 -20424.606,E2 -20424.606} C_VEL
LIN {X 0,Y 218.657,Z 612.134,A -85,B 0,C 180,E1 -20428.158,E2 -20428.158} C_VEL
LIN {X 0,Y 218.656,Z 612.146,A -85,B 0,C 180,E1 -20431.842,E2 -20431.842} C_VEL
LIN {X 0,Y 218.847,Z 611.031,A -85,B 0,C 180,E1 -20435.528,E2 -20435.528} C_VEL
LIN {X 0,Y 219.434,Z 608.787,A -85,B 0,C 180,E1 -20439.215,E2 -20439.215} C_VEL
LIN {X 0,Y 220.537,Z 605.357,A -85,B 0,C 180,E1 -20442.889,E2 -20442.889} C_VEL
LIN {X 0,Y 222.365,Z 600.654,A -85,B 0,C 180,E1 -20446.526,E2 -20446.526} C_VEL
LIN {X 0,Y 224.789,Z 594.558,A -85,B 0,C 180,E1 -20450.115,E2 -20450.115} C_VEL
LIN {X 0,Y 227.921,Z 586.878,A -85,B 0,C 180,E1 -20453.631,E2 -20453.631} C_VEL
LIN {X 0,Y 231.289,Z 578.684,A -85,B 0,C 180,E1 -20456.627,E2 -20456.627} C_VEL
LIN {X 0,Y 235.206,Z 568.941,A -85,B 0,C 180,E1 -20459.495,E2 -20459.495} C_VEL
LIN {X 0,Y 238.957,Z 558.679,A -85,B 0,C 180,E1 -20461.964,E2 -20461.964} C_VEL
LIN {X 0,Y 243.233,Z 546.608,A -85,B 0,C 180,E1 -20464.293,E2 -20464.293} C_VEL
LIN {X 0,Y 246.598,Z 535.787,A -85,B 0,C 180,E1 -20466,E2 -20466} C_VEL
LIN {X 0,Y 250.132,Z 522.917,A -85,B 0,C 180,E1 -20467.669,E2 -20467.669} C_VEL
LIN {X 0,Y 253.23,Z 509.564,A -85,B 0,C 180,E1 -20469.051,E2 -20469.051} C_VEL
LIN {X 0,Y 255.882,Z 495.385,A -85,B 0,C 180,E1 -20470.198,E2 -20470.198} C_VEL
LIN {X 0,Y 258.055,Z 480.602,A -85,B 0,C 180,E1 -20471.073,E2 -20471.073} C_VEL
LIN {X 0,Y 259.601,Z 465.447,A -85,B 0,C 180,E1 -20471.678,E2 -20471.678} C_VEL
LIN {X 0,Y 264.07,Z 386.066,A -85,B 0,C 180,E1 -20473.718,E2 -20473.718} C_VEL
LIN {X 0,Y 264.458,Z 378.226,A -85,B 0,C 180,E1 -20473.927,E2 -20473.927} C_VEL
LIN {X 0,Y 258.599,Z 365.484,A -85,B 0,C 180,E1 -20475.695,E2 -20475.695} C_VEL
LIN {X 0,Y 253.106,Z 355.919,A -85,B 0,C 180,E1 -20477.385,E2 -20477.385} C_VEL
LIN {X 0,Y 244.901,Z 343.127,A -85,B 0,C 180,E1 -20480.1,E2 -20480.1} C_VEL
LIN {X 0,Y 238.743,Z 334.456,A -85,B 0,C 180,E1 -20482.331,E2 -20482.331} C_VEL
LIN {X 0,Y 235.247,Z 329.778,A -85,B 0,C 180,E1 -20483.692,E2 -20483.692} C_VEL
LIN {X 0,Y 232.412,Z 325.942,A -85,B 0,C 180,E1 -20484.863,E2 -20484.863} C_VEL
LIN {X 0,Y 229.763,Z 322.646,A -85,B 0,C 180,E1 -20486,E2 -20486} C_VEL
LIN {X 0,Y 228.81,Z 321.268,A -85,B 0,C 180,E1 -20486.435,E2 -20486.435} C_VEL
LIN {X 0,Y 226.317,Z 318.656,A -85,B 0,C 180,E1 -20487.557,E2 -20487.557} C_VEL
LIN {X 0,Y 224.862,Z 316.132,A -85,B 0,C 180,E1 -20488.3,E2 -20488.3} C_VEL
LIN {X 0,Y 222.457,Z 314.295,A -85,B 0,C 180,E1 -20489.439,E2 -20489.439} C_VEL
LIN {X 0,Y 221.161,Z 312.008,A -85,B 0,C 180,E1 -20490.164,E2 -20490.164} C_VEL
LIN {X 0,Y 220.85,Z 310.567,A -85,B 0,C 180,E1 -20490.445,E2 -20490.445} C_VEL
LIN {X 0,Y 220.88,Z 310.59,A -85,B 0,C 180,E1 -20493.547,E2 -20493.547} C_VEL
LIN {X 0,Y 220.857,Z 310.591,A -85,B 0,C 180,E1 -20497.551,E2 -20497.551} C_VEL
LIN {X 0,Y 220.924,Z 310.579,A -85,B 0,C 180,E1 -20502.617,E2 -20502.617} C_VEL
LIN {X 0,Y 220.988,Z 310.571,A -85,B 0,C 180,E1 -20507.137,E2 -20507.137} C_VEL
LIN {X 0,Y 221.193,Z 310.544,A -85,B 0,C 180,E1 -20510.859,E2 -20510.859} C_VEL
LIN {X 0,Y 221.241,Z 310.549,A -85,B 0,C 180,E1 -20512.7,E2 -20512.7} C_VEL
LIN {X 0,Y 221.467,Z 310.524,A -85,B 0,C 180,E1 -20518.181,E2 -20518.181} C_VEL
LIN {X 0,Y 221.563,Z 310.497,A -85,B 0,C 180,E1 -20520,E2 -20520} C_VEL
LIN {X 0,Y 221.463,Z 310.522,A -85,B 0,C 180,E1 -20521.818,E2 -20521.818} C_VEL
LIN {X 0,Y 221.239,Z 310.552,A -85,B 0,C 180,E1 -20527.3,E2 -20527.3} C_VEL
LIN {X 0,Y 221.056,Z 310.575,A -85,B 0,C 180,E1 -20530.997,E2 -20530.997} C_VEL
LIN {X 0,Y 220.985,Z 310.575,A -85,B 0,C 180,E1 -20532.038,E2 -20532.038} C_VEL
LIN {X 0,Y 220.274,Z 310.664,A -85,B 0,C 180,E1 -20533.56,E2 -20533.56} C_VEL
LIN {X 0,Y 217.357,Z 311.038,A -85,B 0,C 180,E1 -20536.042,E2 -20536.042} C_VEL
LIN {X 0,Y 214.892,Z 311.341,A -85,B 0,C 180,E1 -20538.069,E2 -20538.069} C_VEL
LIN {X 0,Y 213.834,Z 311.477,A -85,B 0,C 180,E1 -20539.645,E2 -20539.645} C_VEL
LIN {X 0,Y 213.747,Z 311.476,A -85,B 0,C 180,E1 -20540.179,E2 -20540.179} C_VEL
LIN {X 0,Y 213.779,Z 311.478,A -85,B 0,C 180,E1 -20543.235,E2 -20543.235} C_VEL
LIN {X 0,Y 213.783,Z 311.483,A -85,B 0,C 180,E1 -20545.757,E2 -20545.757} C_VEL
LIN {X 0,Y 214.504,Z 313.746,A -85,B 0,C 180,E1 -20546.317,E2 -20546.317} C_VEL
LIN {X 0,Y 216.343,Z 316.114,A -85,B 0,C 180,E1 -20547.444,E2 -20547.444} C_VEL
LIN {X 0,Y 218.366,Z 317.535,A -85,B 0,C 180,E1 -20548.538,E2 -20548.538} C_VEL
LIN {X 0,Y 220.166,Z 320.584,A -85,B 0,C 180,E1 -20549.578,E2 -20549.578} C_VEL
LIN {X 0,Y 222.78,Z 323.051,A -85,B 0,C 180,E1 -20550.885,E2 -20550.885} C_VEL
LIN {X 0,Y 225.115,Z 326.399,A -85,B 0,C 180,E1 -20552.055,E2 -20552.055} C_VEL
LIN {X 0,Y 227.738,Z 329.906,A -85,B 0,C 180,E1 -20553.283,E2 -20553.283} C_VEL
LIN {X 0,Y 231.707,Z 335.937,A -85,B 0,C 180,E1 -20555.059,E2 -20555.059} C_VEL
LIN {X 0,Y 234.986,Z 341.01,A -85,B 0,C 180,E1 -20556.431,E2 -20556.431} C_VEL
LIN {X 0,Y 242.223,Z 353.13,A -85,B 0,C 180,E1 -20559.234,E2 -20559.234} C_VEL
LIN {X 0,Y 248.83,Z 365.682,A -85,B 0,C 180,E1 -20561.586,E2 -20561.586} C_VEL
LIN {X 0,Y 255.086,Z 379.024,A -85,B 0,C 180,E1 -20563.67,E2 -20563.67} C_VEL
LIN {X 0,Y 258.985,Z 388.322,A -85,B 0,C 180,E1 -20564.919,E2 -20564.919} C_VEL
LIN {X 0,Y 253.71,Z 478.28,A -85,B 0,C 180,E1 -20567.262,E2 -20567.262} C_VEL
LIN {X 0,Y 251.859,Z 493.619,A -85,B 0,C 180,E1 -20567.89,E2 -20567.89} C_VEL
LIN {X 0,Y 249.314,Z 508.49,A -85,B 0,C 180,E1 -20568.783,E2 -20568.783} C_VEL
LIN {X 0,Y 246.08,Z 523.427,A -85,B 0,C 180,E1 -20570.016,E2 -20570.016} C_VEL
LIN {X 0,Y 242.32,Z 537.585,A -85,B 0,C 180,E1 -20571.543,E2 -20571.543} C_VEL
LIN {X 0,Y 238.413,Z 550.604,A -85,B 0,C 180,E1 -20573.351,E2 -20573.351} C_VEL
LIN {X 0,Y 234.057,Z 563.024,A -85,B 0,C 180,E1 -20575.477,E2 -20575.477} C_VEL
LIN {X 0,Y 229.408,Z 575.205,A -85,B 0,C 180,E1 -20578.1,E2 -20578.1} C_VEL
LIN {X 0,Y 225.192,Z 585.613,A -85,B 0,C 180,E1 -20580.909,E2 -20580.909} C_VEL
LIN {X 0,Y 221.39,Z 595.091,A -85,B 0,C 180,E1 -20584.12,E2 -20584.12} C_VEL
LIN {X 0,Y 218.156,Z 602.594,A -85,B 0,C 180,E1 -20587.258,E2 -20587.258} C_VEL
LIN {X 0,Y 215.361,Z 609.601,A -85,B 0,C 180,E1 -20590.954,E2 -20590.954} C_VEL
LIN {X 0,Y 213.416,Z 615.12,A -85,B 0,C 180,E1 -20594.726,E2 -20594.726} C_VEL
LIN {X 0,Y 212.103,Z 619.296,A -85,B 0,C 180,E1 -20598.533,E2 -20598.533} C_VEL
LIN {X 0,Y 211.519,Z 622.232,A -85,B 0,C 180,E1 -20602.363,E2 -20602.363} C_VEL
LIN {X 0,Y 211.349,Z 623.985,A -85,B 0,C 180,E1 -20606.187,E2 -20606.187} C_VEL
LIN {X 0,Y 211.544,Z 624.59,A -85,B 0,C 180,E1 -20610,E2 -20610} C_VEL
LIN {X 0,Y 211.356,Z 623.921,A -85,B 0,C 180,E1 -20614.006,E2 -20614.006} C_VEL
LIN {X 0,Y 211.483,Z 622.198,A -85,B 0,C 180,E1 -20617.639,E2 -20617.639} C_VEL
LIN {X 0,Y 212.098,Z 619.25,A -85,B 0,C 180,E1 -20621.467,E2 -20621.467} C_VEL
LIN {X 0,Y 213.382,Z 615.061,A -85,B 0,C 180,E1 -20625.277,E2 -20625.277} C_VEL
LIN {X 0,Y 215.294,Z 609.519,A -85,B 0,C 180,E1 -20629.052,E2 -20629.052} C_VEL
LIN {X 0,Y 218.178,Z 602.486,A -85,B 0,C 180,E1 -20632.739,E2 -20632.739} C_VEL
LIN {X 0,Y 221.404,Z 594.971,A -85,B 0,C 180,E1 -20635.878,E2 -20635.878} C_VEL
LIN {X 0,Y 225.352,Z 585.199,A -85,B 0,C 180,E1 -20639.164,E2 -20639.164} C_VEL
LIN {X 0,Y 229.4,Z 575.03,A -85,B 0,C 180,E1 -20641.902,E2 -20641.902} C_VEL
LIN {X 0,Y 234.014,Z 562.803,A -85,B 0,C 180,E1 -20644.53,E2 -20644.53} C_VEL
LIN {X 0,Y 237.986,Z 551.572,A -85,B 0,C 180,E1 -20646.463,E2 -20646.463} C_VEL
LIN {X 0,Y 242.173,Z 537.667,A -85,B 0,C 180,E1 -20648.413,E2 -20648.413} C_VEL
LIN {X 0,Y 246.046,Z 522.997,A -85,B 0,C 180,E1 -20649.991,E2 -20649.991} C_VEL
LIN {X 0,Y 249.101,Z 509.204,A -85,B 0,C 180,E1 -20651.125,E2 -20651.125} C_VEL
LIN {X 0,Y 251.795,Z 493.755,A -85,B 0,C 180,E1 -20652.056,E2 -20652.056} C_VEL
LIN {X 0,Y 253.545,Z 478.455,A -85,B 0,C 180,E1 -20652.705,E2 -20652.705} C_VEL
LIN {X 0,Y 258.055,Z 402.799,A -85,B 0,C 180,E1 -20654.671,E2 -20654.671} C_VEL
LIN {X 0,Y 258.774,Z 388.008,A -85,B 0,C 180,E1 -20655.079,E2 -20655.079} C_VEL
LIN {X 0,Y 253.154,Z 374.777,A -85,B 0,C 180,E1 -20656.892,E2 -20656.892} C_VEL
LIN {X 0,Y 246.057,Z 360.365,A -85,B 0,C 180,E1 -20659.299,E2 -20659.299} C_VEL
LIN {X 0,Y 239.509,Z 348.559,A -85,B 0,C 180,E1 -20661.694,E2 -20661.694} C_VEL
LIN {X 0,Y 233.223,Z 338.235,A -85,B 0,C 180,E1 -20664.203,E2 -20664.203} C_VEL
LIN {X 0,Y 229.42,Z 332.55,A -85,B 0,C 180,E1 -20665.837,E2 -20665.837} C_VEL
LIN {X 0,Y 226.416,Z 328.025,A -85,B 0,C 180,E1 -20667.222,E2 -20667.222} C_VEL
LIN {X 0,Y 222.997,Z 323.509,A -85,B 0,C 180,E1 -20668.873,E2 -20668.873} C_VEL
LIN {X 0,Y 222.324,Z 322.472,A -85,B 0,C 180,E1 -20669.222,E2 -20669.222} C_VEL
LIN {X 0,Y 219.782,Z 320.113,A -85,B 0,C 180,E1 -20670.496,E2 -20670.496} C_VEL
LIN {X 0,Y 218.08,Z 317.139,A -85,B 0,C 180,E1 -20671.487,E2 -20671.487} C_VEL
LIN {X 0,Y 215.675,Z 315.482,A -85,B 0,C 180,E1 -20672.792,E2 -20672.792} C_VEL
LIN {X 0,Y 214.155,Z 313.006,A -85,B 0,C 180,E1 -20673.768,E2 -20673.768} C_VEL
LIN {X 0,Y 213.769,Z 311.481,A -85,B 0,C 180,E1 -20674.176,E2 -20674.176} C_VEL
LIN {X 0,Y 213.769,Z 311.464,A -85,B 0,C 180,E1 -20678.799,E2 -20678.799} C_VEL
LIN {X 0,Y 213.877,Z 311.441,A -85,B 0,C 180,E1 -20682.798,E2 -20682.798} C_VEL
LIN {X 0,Y 213.924,Z 311.429,A -85,B 0,C 180,E1 -20686.705,E2 -20686.705} C_VEL
LIN {X 0,Y 214.117,Z 311.41,A -85,B 0,C 180,E1 -20690.554,E2 -20690.554} C_VEL
LIN {X 0,Y 214.065,Z 311.434,A -85,B 0,C 180,E1 -20694.348,E2 -20694.348} C_VEL
LIN {X 0,Y 214.399,Z 311.393,A -85,B 0,C 180,E1 -20698.122,E2 -20698.122} C_VEL
LIN {X 0,Y 214.503,Z 311.387,A -85,B 0,C 180,E1 -20700,E2 -20700} C_VEL
LIN {X 0,Y 214.4,Z 311.395,A -85,B 0,C 180,E1 -20701.879,E2 -20701.879} C_VEL
LIN {X 0,Y 214.179,Z 311.422,A -85,B 0,C 180,E1 -20707.542,E2 -20707.542} C_VEL
LIN {X 0,Y 213.98,Z 311.446,A -85,B 0,C 180,E1 -20711.366,E2 -20711.366} C_VEL
LIN {X 0,Y 213.876,Z 311.459,A -85,B 0,C 180,E1 -20715.241,E2 -20715.241} C_VEL
LIN {X 0,Y 213.79,Z 311.446,A -85,B 0,C 180,E1 -20719.192,E2 -20719.192} C_VEL
LIN {X 0,Y 213.79,Z 311.467,A -85,B 0,C 180,E1 -20723.234,E2 -20723.234} C_VEL
LIN {X 0,Y 213.853,Z 311.498,A -85,B 0,C 180,E1 -20726.404,E2 -20726.404} C_VEL
LIN {X 0,Y 214.568,Z 313.81,A -85,B 0,C 180,E1 -20726.959,E2 -20726.959} C_VEL
LIN {X 0,Y 216.249,Z 316.004,A -85,B 0,C 180,E1 -20727.983,E2 -20727.983} C_VEL
LIN {X 0,Y 218.293,Z 317.313,A -85,B 0,C 180,E1 -20729.074,E2 -20729.074} C_VEL
LIN {X 0,Y 220.093,Z 320.51,A -85,B 0,C 180,E1 -20730.119,E2 -20730.119} C_VEL
LIN {X 0,Y 222.754,Z 323.085,A -85,B 0,C 180,E1 -20731.445,E2 -20731.445} C_VEL
LIN {X 0,Y 225.333,Z 326.662,A -85,B 0,C 180,E1 -20732.72,E2 -20732.72} C_VEL
LIN {X 0,Y 226.792,Z 328.216,A -85,B 0,C 180,E1 -20733.382,E2 -20733.382} C_VEL
LIN {X 0,Y 229.693,Z 331.992,A -85,B 0,C 180,E1 -20734.679,E2 -20734.679} C_VEL
LIN {X 0,Y 234.384,Z 338.519,A -85,B 0,C 180,E1 -20736.648,E2 -20736.648} C_VEL
LIN {X 0,Y 239.43,Z 345.513,A -85,B 0,C 180,E1 -20738.586,E2 -20738.586} C_VEL
LIN {X 0,Y 248.096,Z 358.965,A -85,B 0,C 180,E1 -20741.629,E2 -20741.629} C_VEL
LIN {X 0,Y 254.062,Z 369.413,A -85,B 0,C 180,E1 -20743.556,E2 -20743.556} C_VEL
LIN {X 0,Y 259.21,Z 380.684,A -85,B 0,C 180,E1 -20745.183,E2 -20745.183} C_VEL
LIN {X 0,Y 254.075,Z 468.184,A -85,B 0,C 180,E1 -20747.472,E2 -20747.472} C_VEL
LIN {X 0,Y 252.297,Z 483.315,A -85,B 0,C 180,E1 -20748.114,E2 -20748.114} C_VEL
LIN {X 0,Y 249.984,Z 498.034,A -85,B 0,C 180,E1 -20749.051,E2 -20749.051} C_VEL
LIN {X 0,Y 246.877,Z 513.106,A -85,B 0,C 180,E1 -20750.346,E2 -20750.346} C_VEL
LIN {X 0,Y 243.501,Z 526.93,A -85,B 0,C 180,E1 -20751.909,E2 -20751.909} C_VEL
LIN {X 0,Y 239.742,Z 539.135,A -85,B 0,C 180,E1 -20753.587,E2 -20753.587} C_VEL
LIN {X 0,Y 235.635,Z 551.538,A -85,B 0,C 180,E1 -20755.74,E2 -20755.74} C_VEL
LIN {X 0,Y 231.525,Z 562.281,A -85,B 0,C 180,E1 -20758.016,E2 -20758.016} C_VEL
LIN {X 0,Y 228.011,Z 571.551,A -85,B 0,C 180,E1 -20760.452,E2 -20760.452} C_VEL
LIN {X 0,Y 223.984,Z 580.99,A -85,B 0,C 180,E1 -20763.441,E2 -20763.441} C_VEL
LIN {X 0,Y 220.1,Z 589.843,A -85,B 0,C 180,E1 -20766.974,E2 -20766.974} C_VEL
LIN {X 0,Y 217.367,Z 596.169,A -85,B 0,C 180,E1 -20770.155,E2 -20770.155} C_VEL
LIN {X 0,Y 214.972,Z 601.974,A -85,B 0,C 180,E1 -20773.866,E2 -20773.866} C_VEL
LIN {X 0,Y 213.639,Z 605.408,A -85,B 0,C 180,E1 -20776.687,E2 -20776.687} C_VEL
LIN {X 0,Y 212.485,Z 608.88,A -85,B 0,C 180,E1 -20780.481,E2 -20780.481} C_VEL
LIN {X 0,Y 211.74,Z 611.35,A -85,B 0,C 180,E1 -20784.717,E2 -20784.717} C_VEL
LIN {X 0,Y 211.558,Z 612.337,A -85,B 0,C 180,E1 -20788.096,E2 -20788.096} C_VEL
LIN {X 0,Y 211.577,Z 612.491,A -85,B 0,C 180,E1 -20790,E2 -20790} C_VEL
LIN {X 0,Y 211.619,Z 611.93,A -85,B 0,C 180,E1 -20793.808,E2 -20793.808} C_VEL
LIN {X 0,Y 212.05,Z 610.255,A -85,B 0,C 180,E1 -20797.618,E2 -20797.618} C_VEL
LIN {X 0,Y 212.932,Z 607.427,A -85,B 0,C 180,E1 -20801.422,E2 -20801.422} C_VEL
LIN {X 0,Y 214.392,Z 603.376,A -85,B 0,C 180,E1 -20805.203,E2 -20805.203} C_VEL
LIN {X 0,Y 216.68,Z 597.994,A -85,B 0,C 180,E1 -20808.926,E2 -20808.926} C_VEL
LIN {X 0,Y 219.598,Z 591.135,A -85,B 0,C 180,E1 -20812.584,E2 -20812.584} C_VEL
LIN {X 0,Y 223.359,Z 582.564,A -85,B 0,C 180,E1 -20816.136,E2 -20816.136} C_VEL
LIN {X 0,Y 227.323,Z 573.445,A -85,B 0,C 180,E1 -20819.138,E2 -20819.138} C_VEL
LIN {X 0,Y 230.832,Z 564.324,A -85,B 0,C 180,E1 -20821.629,E2 -20821.629} C_VEL
LIN {X 0,Y 235.146,Z 553.118,A -85,B 0,C 180,E1 -20824.082,E2 -20824.082} C_VEL
LIN {X 0,Y 239.234,Z 541.023,A -85,B 0,C 180,E1 -20826.242,E2 -20826.242} C_VEL
LIN {X 0,Y 243.315,Z 527.732,A -85,B 0,C 180,E1 -20828.125,E2 -20828.125} C_VEL
LIN {X 0,Y 246.89,Z 513.585,A -85,B 0,C 180,E1 -20829.729,E2 -20829.729} C_VEL
LIN {X 0,Y 250.056,Z 498.16,A -85,B 0,C 180,E1 -20831.068,E2 -20831.068} C_VEL
LIN {X 0,Y 252.539,Z 482.619,A -85,B 0,C 180,E1 -20832.038,E2 -20832.038} C_VEL
LIN {X 0,Y 254.288,Z 467.13,A -85,B 0,C 180,E1 -20832.685,E2 -20832.685} C_VEL
LIN {X 0,Y 259.246,Z 382.178,A -85,B 0,C 180,E1 -20834.902,E2 -20834.902} C_VEL
LIN {X 0,Y 259.237,Z 380.56,A -85,B 0,C 180,E1 -20834.967,E2 -20834.967} C_VEL
LIN {X 0,Y 253.72,Z 368.519,A -85,B 0,C 180,E1 -20836.719,E2 -20836.719} C_VEL
LIN {X 0,Y 246.345,Z 356.067,A -85,B 0,C 180,E1 -20839.127,E2 -20839.127} C_VEL
LIN {X 0,Y 238.669,Z 344.387,A -85,B 0,C 180,E1 -20841.876,E2 -20841.876} C_VEL
LIN {X 0,Y 232.254,Z 335.521,A -85,B 0,C 180,E1 -20844.415,E2 -20844.415} C_VEL
LIN {X 0,Y 229.345,Z 331.594,A -85,B 0,C 180,E1 -20845.664,E2 -20845.664} C_VEL
LIN {X 0,Y 226.581,Z 327.825,A -85,B 0,C 180,E1 -20846.923,E2 -20846.923} C_VEL
LIN {X 0,Y 223.514,Z 324.363,A -85,B 0,C 180,E1 -20848.368,E2 -20848.368} C_VEL
LIN {X 0,Y 222.333,Z 322.464,A -85,B 0,C 180,E1 -20848.986,E2 -20848.986} C_VEL
LIN {X 0,Y 219.746,Z 320.023,A -85,B 0,C 180,E1 -20850.293,E2 -20850.293} C_VEL
LIN {X 0,Y 218.15,Z 317.164,A -85,B 0,C 180,E1 -20851.234,E2 -20851.234} C_VEL
LIN {X 0,Y 215.573,Z 315.354,A -85,B 0,C 180,E1 -20852.646,E2 -20852.646} C_VEL
LIN {X 0,Y 214.164,Z 312.896,A -85,B 0,C 180,E1 -20853.572,E2 -20853.572} C_VEL
LIN {X 0,Y 213.813,Z 311.468,A -85,B 0,C 180,E1 -20853.919,E2 -20853.919} C_VEL
LIN {X 0,Y 213.787,Z 311.47,A -85,B 0,C 180,E1 -20858.8,E2 -20858.8} C_VEL
LIN {X 0,Y 213.887,Z 311.456,A -85,B 0,C 180,E1 -20862.799,E2 -20862.799} C_VEL
LIN {X 0,Y 213.929,Z 311.449,A -85,B 0,C 180,E1 -20866.705,E2 -20866.705} C_VEL
LIN {X 0,Y 214.131,Z 311.424,A -85,B 0,C 180,E1 -20870.555,E2 -20870.555} C_VEL
LIN {X 0,Y 214.076,Z 311.435,A -85,B 0,C 180,E1 -20874.348,E2 -20874.348} C_VEL
LIN {X 0,Y 214.404,Z 311.404,A -85,B 0,C 180,E1 -20878.121,E2 -20878.121} C_VEL
LIN {X 0,Y 214.529,Z 311.373,A -85,B 0,C 180,E1 -20880,E2 -20880} C_VEL
LIN {X 0,Y 214.399,Z 311.402,A -85,B 0,C 180,E1 -20881.878,E2 -20881.878} C_VEL
LIN {X 0,Y 214.18,Z 311.429,A -85,B 0,C 180,E1 -20887.542,E2 -20887.542} C_VEL
LIN {X 0,Y 213.986,Z 311.458,A -85,B 0,C 180,E1 -20891.365,E2 -20891.365} C_VEL
LIN {X 0,Y 213.877,Z 311.469,A -85,B 0,C 180,E1 -20895.241,E2 -20895.241} C_VEL
LIN {X 0,Y 213.789,Z 311.477,A -85,B 0,C 180,E1 -20899.192,E2 -20899.192} C_VEL
LIN {X 0,Y 213.747,Z 311.476,A -85,B 0,C 180,E1 -20900.179,E2 -20900.179} C_VEL
LIN {X 0,Y 213.675,Z 312.075,A -85,B 0,C 180,E1 -20901.768,E2 -20901.768} C_VEL
LIN {X 0,Y 213.648,Z 314.414,A -85,B 0,C 180,E1 -20903.81,E2 -20903.81} C_VEL
LIN {X 0,Y 213.923,Z 317.054,A -85,B 0,C 180,E1 -20905.257,E2 -20905.257} C_VEL
LIN {X 0,Y 215.03,Z 321.432,A -85,B 0,C 180,E1 -20907.031,E2 -20907.031} C_VEL
LIN {X 0,Y 216.034,Z 323.891,A -85,B 0,C 180,E1 -20907.831,E2 -20907.831} C_VEL
LIN {X 0,Y 218.271,Z 327.288,A -85,B 0,C 180,E1 -20909.14,E2 -20909.14} C_VEL
LIN {X 0,Y 220.43,Z 329.453,A -85,B 0,C 180,E1 -20910.261,E2 -20910.261} C_VEL
LIN {X 0,Y 224.986,Z 335.82,A -85,B 0,C 180,E1 -20912.551,E2 -20912.551} C_VEL
LIN {X 0,Y 229.453,Z 342.769,A -85,B 0,C 180,E1 -20914.623,E2 -20914.623} C_VEL
LIN {X 0,Y 232.014,Z 346.878,A -85,B 0,C 180,E1 -20915.736,E2 -20915.736} C_VEL
LIN {X 0,Y 238.608,Z 358.159,A -85,B 0,C 180,E1 -20918.404,E2 -20918.404} C_VEL
LIN {X 0,Y 245.155,Z 370.854,A -85,B 0,C 180,E1 -20920.842,E2 -20920.842} C_VEL
LIN {X 0,Y 251.133,Z 384.059,A -85,B 0,C 180,E1 -20922.93,E2 -20922.93} C_VEL
LIN {X 0,Y 253.848,Z 390.662,A -85,B 0,C 180,E1 -20923.845,E2 -20923.845} C_VEL
LIN {X 0,Y 248.788,Z 475.106,A -85,B 0,C 180,E1 -20926.065,E2 -20926.065} C_VEL
LIN {X 0,Y 247.04,Z 490.687,A -85,B 0,C 180,E1 -20926.661,E2 -20926.661} C_VEL
LIN {X 0,Y 244.547,Z 505.692,A -85,B 0,C 180,E1 -20927.519,E2 -20927.519} C_VEL
LIN {X 0,Y 241.616,Z 519.253,A -85,B 0,C 180,E1 -20928.569,E2 -20928.569} C_VEL
LIN {X 0,Y 237.906,Z 533.412,A -85,B 0,C 180,E1 -20930.003,E2 -20930.003} C_VEL
LIN {X 0,Y 234.011,Z 546.522,A -85,B 0,C 180,E1 -20931.727,E2 -20931.727} C_VEL
LIN {X 0,Y 229.382,Z 559.603,A -85,B 0,C 180,E1 -20933.858,E2 -20933.858} C_VEL
LIN {X 0,Y 224.787,Z 571.448,A -85,B 0,C 180,E1 -20936.293,E2 -20936.293} C_VEL
LIN {X 0,Y 220.652,Z 581.422,A -85,B 0,C 180,E1 -20938.831,E2 -20938.831} C_VEL
LIN {X 0,Y 217.064,Z 589.931,A -85,B 0,C 180,E1 -20941.474,E2 -20941.474} C_VEL
LIN {X 0,Y 213.378,Z 598.261,A -85,B 0,C 180,E1 -20944.649,E2 -20944.649} C_VEL
LIN {X 0,Y 209.965,Z 606.092,A -85,B 0,C 180,E1 -20948.396,E2 -20948.396} C_VEL
LIN {X 0,Y 207.46,Z 612.332,A -85,B 0,C 180,E1 -20952.249,E2 -20952.249} C_VEL
LIN {X 0,Y 205.689,Z 617.164,A -85,B 0,C 180,E1 -20956.162,E2 -20956.162} C_VEL
LIN {X 0,Y 204.697,Z 620.711,A -85,B 0,C 180,E1 -20960.115,E2 -20960.115} C_VEL
LIN {X 0,Y 204.324,Z 623.05,A -85,B 0,C 180,E1 -20964.077,E2 -20964.077} C_VEL
LIN {X 0,Y 204.33,Z 624.229,A -85,B 0,C 180,E1 -20968.029,E2 -20968.029} C_VEL
LIN {X 0,Y 204.462,Z 624.387,A -85,B 0,C 180,E1 -20970,E2 -20970} C_VEL
LIN {X 0,Y 204.259,Z 623.767,A -85,B 0,C 180,E1 -20973.946,E2 -20973.946} C_VEL
LIN {X 0,Y 204.415,Z 621.994,A -85,B 0,C 180,E1 -20977.904,E2 -20977.904} C_VEL
LIN {X 0,Y 205.075,Z 619.044,A -85,B 0,C 180,E1 -20981.866,E2 -20981.866} C_VEL
LIN {X 0,Y 206.45,Z 614.854,A -85,B 0,C 180,E1 -20985.803,E2 -20985.803} C_VEL
LIN {X 0,Y 208.544,Z 609.314,A -85,B 0,C 180,E1 -20989.694,E2 -20989.694} C_VEL
LIN {X 0,Y 211.56,Z 602.279,A -85,B 0,C 180,E1 -20993.492,E2 -20993.492} C_VEL
LIN {X 0,Y 214.983,Z 594.764,A -85,B 0,C 180,E1 -20996.711,E2 -20996.711} C_VEL
LIN {X 0,Y 218.815,Z 585.678,A -85,B 0,C 180,E1 -20999.866,E2 -20999.866} C_VEL
LIN {X 0,Y 223.37,Z 574.823,A -85,B 0,C 180,E1 -21002.87,E2 -21002.87} C_VEL
LIN {X 0,Y 228.142,Z 562.594,A -85,B 0,C 180,E1 -21005.552,E2 -21005.552} C_VEL
LIN {X 0,Y 232.708,Z 550.133,A -85,B 0,C 180,E1 -21007.702,E2 -21007.702} C_VEL
LIN {X 0,Y 236.682,Z 537.268,A -85,B 0,C 180,E1 -21009.509,E2 -21009.509} C_VEL
LIN {X 0,Y 240.63,Z 522.787,A -85,B 0,C 180,E1 -21011.081,E2 -21011.081} C_VEL
LIN {X 0,Y 243.806,Z 508.994,A -85,B 0,C 180,E1 -21012.221,E2 -21012.221} C_VEL
LIN {X 0,Y 246.555,Z 493.541,A -85,B 0,C 180,E1 -21013.165,E2 -21013.165} C_VEL
LIN {X 0,Y 248.383,Z 478.237,A -85,B 0,C 180,E1 -21013.814,E2 -21013.814} C_VEL
LIN {X 0,Y 253.675,Z 391.956,A -85,B 0,C 180,E1 -21016.08,E2 -21016.08} C_VEL
LIN {X 0,Y 253.639,Z 390.275,A -85,B 0,C 180,E1 -21016.155,E2 -21016.155} C_VEL
LIN {X 0,Y 247.937,Z 376.93,A -85,B 0,C 180,E1 -21018.095,E2 -21018.095} C_VEL
LIN {X 0,Y 241.481,Z 363.707,A -85,B 0,C 180,E1 -21020.415,E2 -21020.415} C_VEL
LIN {X 0,Y 235.449,Z 352.781,A -85,B 0,C 180,E1 -21022.744,E2 -21022.744} C_VEL
LIN {X 0,Y 230.092,Z 343.773,A -85,B 0,C 180,E1 -21024.994,E2 -21024.994} C_VEL
LIN {X 0,Y 226.332,Z 337.988,A -85,B 0,C 180,E1 -21026.69,E2 -21026.69} C_VEL
LIN {X 0,Y 223.363,Z 333.463,A -85,B 0,C 180,E1 -21028.124,E2 -21028.124} C_VEL
LIN {X 0,Y 220.242,Z 329.193,A -85,B 0,C 180,E1 -21029.711,E2 -21029.711} C_VEL
LIN {X 0,Y 217.049,Z 325.724,A -85,B 0,C 180,E1 -21031.405,E2 -21031.405} C_VEL
LIN {X 0,Y 215.808,Z 323.656,A -85,B 0,C 180,E1 -21032.153,E2 -21032.153} C_VEL
LIN {X 0,Y 213.211,Z 321.382,A -85,B 0,C 180,E1 -21033.658,E2 -21033.658} C_VEL
LIN {X 0,Y 211.377,Z 318.183,A -85,B 0,C 180,E1 -21034.918,E2 -21034.918} C_VEL
LIN {X 0,Y 208.709,Z 316.478,A -85,B 0,C 180,E1 -21036.658,E2 -21036.658} C_VEL
LIN {X 0,Y 207.093,Z 313.934,A -85,B 0,C 180,E1 -21037.932,E2 -21037.932} C_VEL
LIN {X 0,Y 206.727,Z 312.349,A -85,B 0,C 180,E1 -21038.368,E2 -21038.368} C_VEL
LIN {X 0,Y 206.797,Z 312.315,A -85,B 0,C 180,E1 -21042.19,E2 -21042.19} C_VEL
LIN {X 0,Y 206.866,Z 312.315,A -85,B 0,C 180,E1 -21046.243,E2 -21046.243} C_VEL
LIN {X 0,Y 207.066,Z 312.282,A -85,B 0,C 180,E1 -21050.23,E2 -21050.23} C_VEL
LIN {X 0,Y 207.028,Z 312.31,A -85,B 0,C 180,E1 -21054.155,E2 -21054.155} C_VEL
LIN {X 0,Y 207.338,Z 312.272,A -85,B 0,C 180,E1 -21058.058,E2 -21058.058} C_VEL
LIN {X 0,Y 207.471,Z 312.263,A -85,B 0,C 180,E1 -21060,E2 -21060} C_VEL
LIN {X 0,Y 207.34,Z 312.273,A -85,B 0,C 180,E1 -21061.943,E2 -21061.943} C_VEL
LIN {X 0,Y 207.123,Z 312.302,A -85,B 0,C 180,E1 -21067.801,E2 -21067.801} C_VEL
LIN {X 0,Y 206.901,Z 312.329,A -85,B 0,C 180,E1 -21071.76,E2 -21071.76} C_VEL
LIN {X 0,Y 206.808,Z 312.342,A -85,B 0,C 180,E1 -21075.776,E2 -21075.776} C_VEL
LIN {X 0,Y 206.709,Z 312.321,A -85,B 0,C 180,E1 -21079.877,E2 -21079.877} C_VEL
LIN {X 0,Y 206.748,Z 312.468,A -85,B 0,C 180,E1 -21082.148,E2 -21082.148} C_VEL
LIN {X 0,Y 207.425,Z 314.571,A -85,B 0,C 180,E1 -21082.794,E2 -21082.794} C_VEL
LIN {X 0,Y 209.084,Z 316.812,A -85,B 0,C 180,E1 -21084.052,E2 -21084.052} C_VEL
LIN {X 0,Y 211.567,Z 318.291,A -85,B 0,C 180,E1 -21085.646,E2 -21085.646} C_VEL
LIN {X 0,Y 213.285,Z 321.438,A -85,B 0,C 180,E1 -21086.833,E2 -21086.833} C_VEL
LIN {X 0,Y 216.167,Z 324.156,A -85,B 0,C 180,E1 -21088.507,E2 -21088.507} C_VEL
LIN {X 0,Y 218.481,Z 327.497,A -85,B 0,C 180,E1 -21089.833,E2 -21089.833} C_VEL
LIN {X 0,Y 220.379,Z 329.458,A -85,B 0,C 180,E1 -21090.814,E2 -21090.814} C_VEL
LIN {X 0,Y 223.174,Z 333.15,A -85,B 0,C 180,E1 -21092.227,E2 -21092.227} C_VEL
LIN {X 0,Y 224.74,Z 335.19,A -85,B 0,C 180,E1 -21092.979,E2 -21092.979} C_VEL
LIN {X 0,Y 228.007,Z 339.54,A -85,B 0,C 180,E1 -21094.472,E2 -21094.472} C_VEL
LIN {X 0,Y 233.647,Z 347.342,A -85,B 0,C 180,E1 -21096.85,E2 -21096.85} C_VEL
LIN {X 0,Y 241.078,Z 358.69,A -85,B 0,C 180,E1 -21099.687,E2 -21099.687} C_VEL
LIN {X 0,Y 248.283,Z 370.775,A -85,B 0,C 180,E1 -21102.181,E2 -21102.181} C_VEL
LIN {X 0,Y 252.821,Z 380.129,A -85,B 0,C 180,E1 -21103.692,E2 -21103.692} C_VEL
LIN {X 0,Y 254.059,Z 382.956,A -85,B 0,C 180,E1 -21104.099,E2 -21104.099} C_VEL
LIN {X 0,Y 248.907,Z 468.401,A -85,B 0,C 180,E1 -21106.371,E2 -21106.371} C_VEL
LIN {X 0,Y 247.067,Z 483.528,A -85,B 0,C 180,E1 -21107.016,E2 -21107.016} C_VEL
LIN {X 0,Y 244.664,Z 498.245,A -85,B 0,C 180,E1 -21107.961,E2 -21107.961} C_VEL
LIN {X 0,Y 241.648,Z 512.441,A -85,B 0,C 180,E1 -21109.183,E2 -21109.183} C_VEL
LIN {X 0,Y 237.954,Z 527.138,A -85,B 0,C 180,E1 -21110.854,E2 -21110.854} C_VEL
LIN {X 0,Y 234.067,Z 539.343,A -85,B 0,C 180,E1 -21112.555,E2 -21112.555} C_VEL
LIN {X 0,Y 229.801,Z 551.744,A -85,B 0,C 180,E1 -21114.744,E2 -21114.744} C_VEL
LIN {X 0,Y 225.506,Z 562.488,A -85,B 0,C 180,E1 -21117.056,E2 -21117.056} C_VEL
LIN {X 0,Y 221.843,Z 571.757,A -85,B 0,C 180,E1 -21119.545,E2 -21119.545} C_VEL
LIN {X 0,Y 218.189,Z 579.975,A -85,B 0,C 180,E1 -21122.158,E2 -21122.158} C_VEL
LIN {X 0,Y 214.516,Z 588.049,A -85,B 0,C 180,E1 -21125.31,E2 -21125.31} C_VEL
LIN {X 0,Y 211.425,Z 594.708,A -85,B 0,C 180,E1 -21128.553,E2 -21128.553} C_VEL
LIN {X 0,Y 208.732,Z 600.864,A -85,B 0,C 180,E1 -21132.361,E2 -21132.361} C_VEL
LIN {X 0,Y 206.714,Z 605.613,A -85,B 0,C 180,E1 -21136.232,E2 -21136.232} C_VEL
LIN {X 0,Y 205.463,Z 609.084,A -85,B 0,C 180,E1 -21140.153,E2 -21140.153} C_VEL
LIN {X 0,Y 204.71,Z 611.376,A -85,B 0,C 180,E1 -21144.089,E2 -21144.089} C_VEL
LIN {X 0,Y 204.462,Z 612.54,A -85,B 0,C 180,E1 -21148.03,E2 -21148.03} C_VEL
LIN {X 0,Y 204.496,Z 612.694,A -85,B 0,C 180,E1 -21150,E2 -21150} C_VEL
LIN {X 0,Y 204.539,Z 612.133,A -85,B 0,C 180,E1 -21153.94,E2 -21153.94} C_VEL
LIN {X 0,Y 205.002,Z 610.458,A -85,B 0,C 180,E1 -21157.882,E2 -21157.882} C_VEL
LIN {X 0,Y 205.938,Z 607.631,A -85,B 0,C 180,E1 -21161.815,E2 -21161.815} C_VEL
LIN {X 0,Y 207.516,Z 603.579,A -85,B 0,C 180,E1 -21165.72,E2 -21165.72} C_VEL
LIN {X 0,Y 209.93,Z 598.197,A -85,B 0,C 180,E1 -21169.558,E2 -21169.558} C_VEL
LIN {X 0,Y 213.016,Z 591.338,A -85,B 0,C 180,E1 -21173.322,E2 -21173.322} C_VEL
LIN {X 0,Y 216.999,Z 582.766,A -85,B 0,C 180,E1 -21176.963,E2 -21176.963} C_VEL
LIN {X 0,Y 220.486,Z 575.055,A -85,B 0,C 180,E1 -21179.607,E2 -21179.607} C_VEL
LIN {X 0,Y 224.868,Z 564.362,A -85,B 0,C 180,E1 -21182.623,E2 -21182.623} C_VEL
LIN {X 0,Y 229.668,Z 552.328,A -85,B 0,C 180,E1 -21185.28,E2 -21185.28} C_VEL
LIN {X 0,Y 233.948,Z 540.038,A -85,B 0,C 180,E1 -21187.467,E2 -21187.467} C_VEL
LIN {X 0,Y 238.209,Z 526.464,A -85,B 0,C 180,E1 -21189.369,E2 -21189.369} C_VEL
LIN {X 0,Y 241.662,Z 513.075,A -85,B 0,C 180,E1 -21190.876,E2 -21190.876} C_VEL
LIN {X 0,Y 244.744,Z 498.355,A -85,B 0,C 180,E1 -21192.161,E2 -21192.161} C_VEL
LIN {X 0,Y 247.317,Z 482.81,A -85,B 0,C 180,E1 -21193.138,E2 -21193.138} C_VEL
LIN {X 0,Y 249.113,Z 467.314,A -85,B 0,C 180,E1 -21193.793,E2 -21193.793} C_VEL
LIN {X 0,Y 254.103,Z 384.628,A -85,B 0,C 180,E1 -21195.979,E2 -21195.979} C_VEL
LIN {X 0,Y 254.102,Z 382.918,A -85,B 0,C 180,E1 -21196.048,E2 -21196.048} C_VEL
LIN {X 0,Y 249.354,Z 372.578,A -85,B 0,C 180,E1 -21197.631,E2 -21197.631} C_VEL
LIN {X 0,Y 242.275,Z 360.509,A -85,B 0,C 180,E1 -21200.057,E2 -21200.057} C_VEL
LIN {X 0,Y 235.282,Z 349.666,A -85,B 0,C 180,E1 -21202.684,E2 -21202.684} C_VEL
LIN {X 0,Y 229.021,Z 340.92,A -85,B 0,C 180,E1 -21205.275,E2 -21205.275} C_VEL
LIN {X 0,Y 226.443,Z 337.393,A -85,B 0,C 180,E1 -21206.433,E2 -21206.433} C_VEL
LIN {X 0,Y 223.521,Z 333.438,A -85,B 0,C 180,E1 -21207.822,E2 -21207.822} C_VEL
LIN {X 0,Y 220.692,Z 329.951,A -85,B 0,C 180,E1 -21209.235,E2 -21209.235} C_VEL
LIN {X 0,Y 219.806,Z 328.675,A -85,B 0,C 180,E1 -21209.709,E2 -21209.709} C_VEL
LIN {X 0,Y 217.028,Z 325.634,A -85,B 0,C 180,E1 -21211.204,E2 -21211.204} C_VEL
LIN {X 0,Y 215.792,Z 323.605,A -85,B 0,C 180,E1 -21211.952,E2 -21211.952} C_VEL
LIN {X 0,Y 213.204,Z 321.349,A -85,B 0,C 180,E1 -21213.465,E2 -21213.465} C_VEL
LIN {X 0,Y 211.485,Z 318.174,A -85,B 0,C 180,E1 -21214.668,E2 -21214.668} C_VEL
LIN {X 0,Y 208.836,Z 316.571,A -85,B 0,C 180,E1 -21216.399,E2 -21216.399} C_VEL
LIN {X 0,Y 207.172,Z 314.089,A -85,B 0,C 180,E1 -21217.708,E2 -21217.708} C_VEL
LIN {X 0,Y 206.737,Z 312.347,A -85,B 0,C 180,E1 -21218.237,E2 -21218.237} C_VEL
LIN {X 0,Y 206.82,Z 312.335,A -85,B 0,C 180,E1 -21222.192,E2 -21222.192} C_VEL
LIN {X 0,Y 206.87,Z 312.329,A -85,B 0,C 180,E1 -21226.242,E2 -21226.242} C_VEL
LIN {X 0,Y 207.075,Z 312.305,A -85,B 0,C 180,E1 -21230.23,E2 -21230.23} C_VEL
LIN {X 0,Y 207.039,Z 312.314,A -85,B 0,C 180,E1 -21234.155,E2 -21234.155} C_VEL
LIN {X 0,Y 207.343,Z 312.284,A -85,B 0,C 180,E1 -21238.057,E2 -21238.057} C_VEL
LIN {X 0,Y 207.495,Z 312.249,A -85,B 0,C 180,E1 -21240,E2 -21240} C_VEL
LIN {X 0,Y 207.038,Z 312.309,A -85,B 0,C 180,E1 -21243.893,E2 -21243.893} C_VEL
LIN {X 0,Y 207.124,Z 312.305,A -85,B 0,C 180,E1 -21247.8,E2 -21247.8} C_VEL
LIN {X 0,Y 206.906,Z 312.338,A -85,B 0,C 180,E1 -21251.759,E2 -21251.759} C_VEL
LIN {X 0,Y 206.809,Z 312.354,A -85,B 0,C 180,E1 -21255.775,E2 -21255.775} C_VEL
LIN {X 0,Y 206.71,Z 312.366,A -85,B 0,C 180,E1 -21259.876,E2 -21259.876} C_VEL
LIN {X 0,Y 206.743,Z 312.556,A -85,B 0,C 180,E1 -21261.5,E2 -21261.5} C_VEL
LIN {X 0,Y 207.53,Z 314.875,A -85,B 0,C 180,E1 -21262.247,E2 -21262.247} C_VEL
LIN {X 0,Y 209.701,Z 317.316,A -85,B 0,C 180,E1 -21263.845,E2 -21263.845} C_VEL
LIN {X 0,Y 211.591,Z 318.426,A -85,B 0,C 180,E1 -21265.055,E2 -21265.055} C_VEL
LIN {X 0,Y 213.42,Z 321.622,A -85,B 0,C 180,E1 -21266.315,E2 -21266.315} C_VEL
LIN {X 0,Y 216.034,Z 323.891,A -85,B 0,C 180,E1 -21267.831,E2 -21267.831} C_VEL
LIN {X 0,Y 218.255,Z 329.238,A -85,B 0,C 180,E1 -21269.261,E2 -21269.261} C_VEL
LIN {X 0,Y 222.574,Z 340.78,A -85,B 0,C 180,E1 -21271.869,E2 -21271.869} C_VEL
LIN {X 0,Y 225.145,Z 346.167,A -85,B 0,C 180,E1 -21273.206,E2 -21273.206} C_VEL
LIN {X 0,Y 230.549,Z 355.121,A -85,B 0,C 180,E1 -21275.662,E2 -21275.662} C_VEL
LIN {X 0,Y 237.531,Z 367.978,A -85,B 0,C 180,E1 -21278.545,E2 -21278.545} C_VEL
LIN {X 0,Y 243.781,Z 380.994,A -85,B 0,C 180,E1 -21280.916,E2 -21280.916} C_VEL
LIN {X 0,Y 248.84,Z 393.004,A -85,B 0,C 180,E1 -21282.736,E2 -21282.736} C_VEL
LIN {X 0,Y 243.473,Z 477.907,A -85,B 0,C 180,E1 -21284.993,E2 -21284.993} C_VEL
LIN {X 0,Y 241.517,Z 493.235,A -85,B 0,C 180,E1 -21285.631,E2 -21285.631} C_VEL
LIN {X 0,Y 238.837,Z 508.1,A -85,B 0,C 180,E1 -21286.543,E2 -21286.543} C_VEL
LIN {X 0,Y 235.348,Z 523.031,A -85,B 0,C 180,E1 -21287.788,E2 -21287.788} C_VEL
LIN {X 0,Y 231.598,Z 536.296,A -85,B 0,C 180,E1 -21289.241,E2 -21289.241} C_VEL
LIN {X 0,Y 227.57,Z 548.911,A -85,B 0,C 180,E1 -21291.007,E2 -21291.007} C_VEL
LIN {X 0,Y 222.821,Z 561.548,A -85,B 0,C 180,E1 -21293.183,E2 -21293.183} C_VEL
LIN {X 0,Y 218.111,Z 573.037,A -85,B 0,C 180,E1 -21295.676,E2 -21295.676} C_VEL
LIN {X 0,Y 213.907,Z 582.713,A -85,B 0,C 180,E1 -21298.287,E2 -21298.287} C_VEL
LIN {X 0,Y 210.243,Z 590.987,A -85,B 0,C 180,E1 -21301.008,E2 -21301.008} C_VEL
LIN {X 0,Y 206.409,Z 599.139,A -85,B 0,C 180,E1 -21304.271,E2 -21304.271} C_VEL
LIN {X 0,Y 203.306,Z 605.888,A -85,B 0,C 180,E1 -21307.651,E2 -21307.651} C_VEL
LIN {X 0,Y 200.624,Z 612.128,A -85,B 0,C 180,E1 -21311.623,E2 -21311.623} C_VEL
LIN {X 0,Y 198.758,Z 616.96,A -85,B 0,C 180,E1 -21315.67,E2 -21315.67} C_VEL
LIN {X 0,Y 197.657,Z 620.507,A -85,B 0,C 180,E1 -21319.76,E2 -21319.76} C_VEL
LIN {X 0,Y 197.227,Z 622.847,A -85,B 0,C 180,E1 -21323.863,E2 -21323.863} C_VEL
LIN {X 0,Y 197.234,Z 624.026,A -85,B 0,C 180,E1 -21327.958,E2 -21327.958} C_VEL
LIN {X 0,Y 197.361,Z 624.184,A -85,B 0,C 180,E1 -21330,E2 -21330} C_VEL
LIN {X 0,Y 197.171,Z 623.564,A -85,B 0,C 180,E1 -21334.088,E2 -21334.088} C_VEL
LIN {X 0,Y 197.34,Z 621.789,A -85,B 0,C 180,E1 -21338.19,E2 -21338.19} C_VEL
LIN {X 0,Y 198.066,Z 618.839,A -85,B 0,C 180,E1 -21342.292,E2 -21342.292} C_VEL
LIN {X 0,Y 199.543,Z 614.648,A -85,B 0,C 180,E1 -21346.365,E2 -21346.365} C_VEL
LIN {X 0,Y 201.808,Z 609.107,A -85,B 0,C 180,E1 -21350.38,E2 -21350.38} C_VEL
LIN {X 0,Y 205.014,Z 602.072,A -85,B 0,C 180,E1 -21354.29,E2 -21354.29} C_VEL
LIN {X 0,Y 208.592,Z 594.557,A -85,B 0,C 180,E1 -21357.598,E2 -21357.598} C_VEL
LIN {X 0,Y 212.775,Z 585.174,A -85,B 0,C 180,E1 -21360.923,E2 -21360.923} C_VEL
LIN {X 0,Y 217.406,Z 574.617,A -85,B 0,C 180,E1 -21363.891,E2 -21363.891} C_VEL
LIN {X 0,Y 222.379,Z 562.387,A -85,B 0,C 180,E1 -21366.62,E2 -21366.62} C_VEL
LIN {X 0,Y 227.1,Z 549.925,A -85,B 0,C 180,E1 -21368.804,E2 -21368.804} C_VEL
LIN {X 0,Y 231.338,Z 536.764,A -85,B 0,C 180,E1 -21370.664,E2 -21370.664} C_VEL
LIN {X 0,Y 235.32,Z 522.578,A -85,B 0,C 180,E1 -21372.218,E2 -21372.218} C_VEL
LIN {X 0,Y 238.605,Z 508.784,A -85,B 0,C 180,E1 -21373.365,E2 -21373.365} C_VEL
LIN {X 0,Y 241.304,Z 494.131,A -85,B 0,C 180,E1 -21374.273,E2 -21374.273} C_VEL
LIN {X 0,Y 243.3,Z 478.017,A -85,B 0,C 180,E1 -21374.974,E2 -21374.974} C_VEL
LIN {X 0,Y 248.153,Z 402.028,A -85,B 0,C 180,E1 -21376.991,E2 -21376.991} C_VEL
LIN {X 0,Y 248.721,Z 392.992,A -85,B 0,C 180,E1 -21377.225,E2 -21377.225} C_VEL
LIN {X 0,Y 243.706,Z 381.009,A -85,B 0,C 180,E1 -21379.027,E2 -21379.027} C_VEL
LIN {X 0,Y 237.267,Z 367.592,A -85,B 0,C 180,E1 -21381.468,E2 -21381.468} C_VEL
LIN {X 0,Y 231.065,Z 356.216,A -85,B 0,C 180,E1 -21384.008,E2 -21384.008} C_VEL
LIN {X 0,Y 226.703,Z 348.817,A -85,B 0,C 180,E1 -21385.948,E2 -21385.948} C_VEL
LIN {X 0,Y 223.16,Z 343.243,A -85,B 0,C 180,E1 -21387.63,E2 -21387.63} C_VEL
LIN {X 0,Y 220.363,Z 338.927,A -85,B 0,C 180,E1 -21389.051,E2 -21389.051} C_VEL
LIN {X 0,Y 217.249,Z 334.769,A -85,B 0,C 180,E1 -21390.709,E2 -21390.709} C_VEL
LIN {X 0,Y 214.5,Z 331.512,A -85,B 0,C 180,E1 -21392.261,E2 -21392.261} C_VEL
LIN {X 0,Y 213.49,Z 330.005,A -85,B 0,C 180,E1 -21392.883,E2 -21392.883} C_VEL
LIN {X 0,Y 210.839,Z 327.288,A -85,B 0,C 180,E1 -21394.519,E2 -21394.519} C_VEL
LIN {X 0,Y 209.256,Z 324.745,A -85,B 0,C 180,E1 -21395.64,E2 -21395.64} C_VEL
LIN {X 0,Y 206.669,Z 322.719,A -85,B 0,C 180,E1 -21397.435,E2 -21397.435} C_VEL
LIN {X 0,Y 204.941,Z 319.722,A -85,B 0,C 180,E1 -21398.895,E2 -21398.895} C_VEL
LIN {X 0,Y 204.689,Z 319.141,A -85,B 0,C 180,E1 -21399.132,E2 -21399.132} C_VEL
LIN {X 0,Y 201.888,Z 317.479,A -85,B 0,C 180,E1 -21401.479,E2 -21401.479} C_VEL
LIN {X 0,Y 200.223,Z 315.005,A -85,B 0,C 180,E1 -21403.233,E2 -21403.233} C_VEL
LIN {X 0,Y 199.76,Z 313.216,A -85,B 0,C 180,E1 -21403.915,E2 -21403.915} C_VEL
LIN {X 0,Y 200.018,Z 313.155,A -85,B 0,C 180,E1 -21409.882,E2 -21409.882} C_VEL
LIN {X 0,Y 199.991,Z 313.187,A -85,B 0,C 180,E1 -21413.949,E2 -21413.949} C_VEL
LIN {X 0,Y 200.28,Z 313.151,A -85,B 0,C 180,E1 -21417.989,E2 -21417.989} C_VEL
LIN {X 0,Y 200.439,Z 313.138,A -85,B 0,C 180,E1 -21420,E2 -21420} C_VEL
LIN {X 0,Y 199.99,Z 313.193,A -85,B 0,C 180,E1 -21424.031,E2 -21424.031} C_VEL
LIN {X 0,Y 200.071,Z 313.182,A -85,B 0,C 180,E1 -21428.078,E2 -21428.078} C_VEL
LIN {X 0,Y 199.852,Z 313.21,A -85,B 0,C 180,E1 -21432.181,E2 -21432.181} C_VEL
LIN {X 0,Y 199.751,Z 313.235,A -85,B 0,C 180,E1 -21436.545,E2 -21436.545} C_VEL
LIN {X 0,Y 200.332,Z 315.283,A -85,B 0,C 180,E1 -21437.349,E2 -21437.349} C_VEL
LIN {X 0,Y 202.089,Z 317.711,A -85,B 0,C 180,E1 -21439.16,E2 -21439.16} C_VEL
LIN {X 0,Y 204.902,Z 319.518,A -85,B 0,C 180,E1 -21441.505,E2 -21441.505} C_VEL
LIN {X 0,Y 206.441,Z 322.398,A -85,B 0,C 180,E1 -21442.833,E2 -21442.833} C_VEL
LIN {X 0,Y 208.936,Z 324.559,A -85,B 0,C 180,E1 -21444.6,E2 -21444.6} C_VEL
LIN {X 0,Y 209.638,Z 325.153,A -85,B 0,C 180,E1 -21445.067,E2 -21445.067} C_VEL
LIN {X 0,Y 211.704,Z 328.376,A -85,B 0,C 180,E1 -21446.492,E2 -21446.492} C_VEL
LIN {X 0,Y 213.955,Z 330.564,A -85,B 0,C 180,E1 -21447.844,E2 -21447.844} C_VEL
LIN {X 0,Y 216.594,Z 334.182,A -85,B 0,C 180,E1 -21449.392,E2 -21449.392} C_VEL
LIN {X 0,Y 218.051,Z 335.766,A -85,B 0,C 180,E1 -21450.173,E2 -21450.173} C_VEL
LIN {X 0,Y 221.024,Z 339.624,A -85,B 0,C 180,E1 -21451.72,E2 -21451.72} C_VEL
LIN {X 0,Y 225.778,Z 346.242,A -85,B 0,C 180,E1 -21454.01,E2 -21454.01} C_VEL
LIN {X 0,Y 230.946,Z 353.612,A -85,B 0,C 180,E1 -21456.264,E2 -21456.264} C_VEL
LIN {X 0,Y 237.398,Z 363.633,A -85,B 0,C 180,E1 -21458.831,E2 -21458.831} C_VEL
LIN {X 0,Y 244.345,Z 375.478,A -85,B 0,C 180,E1 -21461.349,E2 -21461.349} C_VEL
LIN {X 0,Y 248.747,Z 384.713,A -85,B 0,C 180,E1 -21462.884,E2 -21462.884} C_VEL
LIN {X 0,Y 249.075,Z 385.518,A -85,B 0,C 180,E1 -21463,E2 -21463} C_VEL
LIN {X 0,Y 243.958,Z 467.259,A -85,B 0,C 180,E1 -21465.18,E2 -21465.18} C_VEL
LIN {X 0,Y 242.044,Z 482.871,A -85,B 0,C 180,E1 -21465.826,E2 -21465.826} C_VEL
LIN {X 0,Y 239.453,Z 498.456,A -85,B 0,C 180,E1 -21466.827,E2 -21466.827} C_VEL
LIN {X 0,Y 236.307,Z 512.745,A -85,B 0,C 180,E1 -21468.069,E2 -21468.069} C_VEL
LIN {X 0,Y 232.489,Z 527.346,A -85,B 0,C 180,E1 -21469.749,E2 -21469.749} C_VEL
LIN {X 0,Y 228.457,Z 539.55,A -85,B 0,C 180,E1 -21471.47,E2 -21471.47} C_VEL
LIN {X 0,Y 224.018,Z 551.952,A -85,B 0,C 180,E1 -21473.691,E2 -21473.691} C_VEL
LIN {X 0,Y 219.717,Z 562.34,A -85,B 0,C 180,E1 -21475.961,E2 -21475.961} C_VEL
LIN {X 0,Y 215.734,Z 571.963,A -85,B 0,C 180,E1 -21478.586,E2 -21478.586} C_VEL
LIN {X 0,Y 211.883,Z 580.181,A -85,B 0,C 180,E1 -21481.253,E2 -21481.253} C_VEL
LIN {X 0,Y 208.063,Z 588.254,A -85,B 0,C 180,E1 -21484.491,E2 -21484.491} C_VEL
LIN {X 0,Y 204.24,Z 596.111,A -85,B 0,C 180,E1 -21488.51,E2 -21488.51} C_VEL
LIN {X 0,Y 201.32,Z 602.383,A -85,B 0,C 180,E1 -21492.739,E2 -21492.739} C_VEL
LIN {X 0,Y 199.786,Z 605.818,A -85,B 0,C 180,E1 -21495.745,E2 -21495.745} C_VEL
LIN {X 0,Y 198.464,Z 609.288,A -85,B 0,C 180,E1 -21499.802,E2 -21499.802} C_VEL
LIN {X 0,Y 197.657,Z 611.579,A -85,B 0,C 180,E1 -21503.877,E2 -21503.877} C_VEL
LIN {X 0,Y 197.369,Z 612.743,A -85,B 0,C 180,E1 -21507.959,E2 -21507.959} C_VEL
LIN {X 0,Y 197.397,Z 612.897,A -85,B 0,C 180,E1 -21510,E2 -21510} C_VEL
LIN {X 0,Y 197.463,Z 612.335,A -85,B 0,C 180,E1 -21514.082,E2 -21514.082} C_VEL
LIN {X 0,Y 197.95,Z 610.661,A -85,B 0,C 180,E1 -21518.164,E2 -21518.164} C_VEL
LIN {X 0,Y 198.967,Z 607.834,A -85,B 0,C 180,E1 -21522.235,E2 -21522.235} C_VEL
LIN {X 0,Y 200.664,Z 603.781,A -85,B 0,C 180,E1 -21526.271,E2 -21526.271} C_VEL
LIN {X 0,Y 203.217,Z 598.4,A -85,B 0,C 180,E1 -21530.232,E2 -21530.232} C_VEL
LIN {X 0,Y 206.488,Z 591.54,A -85,B 0,C 180,E1 -21534.106,E2 -21534.106} C_VEL
LIN {X 0,Y 210.662,Z 582.968,A -85,B 0,C 180,E1 -21537.843,E2 -21537.843} C_VEL
LIN {X 0,Y 214.335,Z 575.256,A -85,B 0,C 180,E1 -21540.546,E2 -21540.546} C_VEL
LIN {X 0,Y 218.9,Z 564.563,A -85,B 0,C 180,E1 -21543.629,E2 -21543.629} C_VEL
LIN {X 0,Y 223.913,Z 552.527,A -85,B 0,C 180,E1 -21546.329,E2 -21546.329} C_VEL
LIN {X 0,Y 228.364,Z 540.237,A -85,B 0,C 180,E1 -21548.549,E2 -21548.549} C_VEL
LIN {X 0,Y 232.762,Z 526.661,A -85,B 0,C 180,E1 -21550.478,E2 -21550.478} C_VEL
LIN {X 0,Y 236.488,Z 512.672,A -85,B 0,C 180,E1 -21552.059,E2 -21552.059} C_VEL
LIN {X 0,Y 239.535,Z 498.55,A -85,B 0,C 180,E1 -21553.299,E2 -21553.299} C_VEL
LIN {X 0,Y 242.198,Z 483,A -85,B 0,C 180,E1 -21554.284,E2 -21554.284} C_VEL
LIN {X 0,Y 244.054,Z 467.496,A -85,B 0,C 180,E1 -21554.943,E2 -21554.943} C_VEL
LIN {X 0,Y 249.142,Z 386.427,A -85,B 0,C 180,E1 -21557.105,E2 -21557.105} C_VEL
LIN {X 0,Y 248.865,Z 384.821,A -85,B 0,C 180,E1 -21557.242,E2 -21557.242} C_VEL
LIN {X 0,Y 244.656,Z 375.873,A -85,B 0,C 180,E1 -21558.715,E2 -21558.715} C_VEL
LIN {X 0,Y 236.918,Z 362.694,A -85,B 0,C 180,E1 -21561.536,E2 -21561.536} C_VEL
LIN {X 0,Y 229.936,Z 352.003,A -85,B 0,C 180,E1 -21564.357,E2 -21564.357} C_VEL
LIN {X 0,Y 223.786,Z 343.374,A -85,B 0,C 180,E1 -21567.13,E2 -21567.13} C_VEL
LIN {X 0,Y 220.519,Z 339.079,A -85,B 0,C 180,E1 -21568.742,E2 -21568.742} C_VEL
LIN {X 0,Y 217.281,Z 334.777,A -85,B 0,C 180,E1 -21570.472,E2 -21570.472} C_VEL
LIN {X 0,Y 214.443,Z 331.323,A -85,B 0,C 180,E1 -21572.092,E2 -21572.092} C_VEL
LIN {X 0,Y 213.499,Z 329.953,A -85,B 0,C 180,E1 -21572.677,E2 -21572.677} C_VEL
LIN {X 0,Y 210.928,Z 327.385,A -85,B 0,C 180,E1 -21574.27,E2 -21574.27} C_VEL
LIN {X 0,Y 209.455,Z 324.822,A -85,B 0,C 180,E1 -21575.334,E2 -21575.334} C_VEL
LIN {X 0,Y 206.856,Z 322.89,A -85,B 0,C 180,E1 -21577.135,E2 -21577.135} C_VEL
LIN {X 0,Y 205.058,Z 319.97,A -85,B 0,C 180,E1 -21578.644,E2 -21578.644} C_VEL
LIN {X 0,Y 204.53,Z 319.099,A -85,B 0,C 180,E1 -21579.114,E2 -21579.114} C_VEL
LIN {X 0,Y 201.788,Z 317.409,A -85,B 0,C 180,E1 -21581.469,E2 -21581.469} C_VEL
LIN {X 0,Y 200.121,Z 314.775,A -85,B 0,C 180,E1 -21583.289,E2 -21583.289} C_VEL
LIN {X 0,Y 199.788,Z 313.22,A -85,B 0,C 180,E1 -21583.917,E2 -21583.917} C_VEL
LIN {X 0,Y 200.018,Z 313.186,A -85,B 0,C 180,E1 -21589.881,E2 -21589.881} C_VEL
LIN {X 0,Y 200.002,Z 313.192,A -85,B 0,C 180,E1 -21593.948,E2 -21593.948} C_VEL
LIN {X 0,Y 200.285,Z 313.163,A -85,B 0,C 180,E1 -21597.989,E2 -21597.989} C_VEL
LIN {X 0,Y 200.459,Z 313.125,A -85,B 0,C 180,E1 -21600,E2 -21600} C_VEL
LIN {X 0,Y 199.984,Z 313.187,A -85,B 0,C 180,E1 -21604.03,E2 -21604.03} C_VEL
LIN {X 0,Y 200.072,Z 313.18,A -85,B 0,C 180,E1 -21608.077,E2 -21608.077} C_VEL
LIN {X 0,Y 199.855,Z 313.211,A -85,B 0,C 180,E1 -21612.18,E2 -21612.18} C_VEL
LIN {X 0,Y 199.772,Z 313.268,A -85,B 0,C 180,E1 -21615.822,E2 -21615.822} C_VEL
LIN {X 0,Y 200.387,Z 315.432,A -85,B 0,C 180,E1 -21616.687,E2 -21616.687} C_VEL
LIN {X 0,Y 202.648,Z 318.168,A -85,B 0,C 180,E1 -21618.973,E2 -21618.973} C_VEL
LIN {X 0,Y 204.841,Z 319.396,A -85,B 0,C 180,E1 -21620.786,E2 -21620.786} C_VEL
LIN {X 0,Y 206.31,Z 322.229,A -85,B 0,C 180,E1 -21622.082,E2 -21622.082} C_VEL
LIN {X 0,Y 208.721,Z 324.45,A -85,B 0,C 180,E1 -21623.832,E2 -21623.832} C_VEL
LIN {X 0,Y 209.654,Z 325.206,A -85,B 0,C 180,E1 -21624.459,E2 -21624.459} C_VEL
LIN {X 0,Y 211.83,Z 328.497,A -85,B 0,C 180,E1 -21625.962,E2 -21625.962} C_VEL
LIN {X 0,Y 213.971,Z 330.572,A -85,B 0,C 180,E1 -21627.255,E2 -21627.255} C_VEL
LIN {X 0,Y 216.711,Z 334.289,A -85,B 0,C 180,E1 -21628.869,E2 -21628.869} C_VEL
LIN {X 0,Y 218.107,Z 335.831,A -85,B 0,C 180,E1 -21629.623,E2 -21629.623} C_VEL
LIN {X 0,Y 222.343,Z 341.799,A -85,B 0,C 180,E1 -21631.835,E2 -21631.835} C_VEL
LIN {X 0,Y 225.145,Z 346.167,A -85,B 0,C 180,E1 -21633.206,E2 -21633.206} C_VEL
LIN {X 0,Y 226.984,Z 350.417,A -85,B 0,C 180,E1 -21634.139,E2 -21634.139} C_VEL
LIN {X 0,Y 230.931,Z 365.561,A -85,B 0,C 180,E1 -21636.331,E2 -21636.331} C_VEL
LIN {X 0,Y 232.609,Z 370.307,A -85,B 0,C 180,E1 -21637.123,E2 -21637.123} C_VEL
LIN {X 0,Y 233.301,Z 371.742,A -85,B 0,C 180,E1 -21637.416,E2 -21637.416} C_VEL
LIN {X 0,Y 238.938,Z 383.515,A -85,B 0,C 180,E1 -21639.683,E2 -21639.683} C_VEL
LIN {X 0,Y 243.923,Z 395.354,A -85,B 0,C 180,E1 -21641.58,E2 -21641.58} C_VEL
LIN {X 0,Y 238.498,Z 477.72,A -85,B 0,C 180,E1 -21643.785,E2 -21643.785} C_VEL
LIN {X 0,Y 236.501,Z 493.043,A -85,B 0,C 180,E1 -21644.43,E2 -21644.43} C_VEL
LIN {X 0,Y 233.732,Z 507.905,A -85,B 0,C 180,E1 -21645.345,E2 -21645.345} C_VEL
LIN {X 0,Y 230.132,Z 522.834,A -85,B 0,C 180,E1 -21646.598,E2 -21646.598} C_VEL
LIN {X 0,Y 225.998,Z 536.917,A -85,B 0,C 180,E1 -21648.162,E2 -21648.162} C_VEL
LIN {X 0,Y 221.621,Z 550.005,A -85,B 0,C 180,E1 -21650.048,E2 -21650.048} C_VEL
LIN {X 0,Y 216.726,Z 562.42,A -85,B 0,C 180,E1 -21652.261,E2 -21652.261} C_VEL
LIN {X 0,Y 211.494,Z 574.599,A -85,B 0,C 180,E1 -21655.026,E2 -21655.026} C_VEL
LIN {X 0,Y 206.494,Z 585.365,A -85,B 0,C 180,E1 -21658.13,E2 -21658.13} C_VEL
LIN {X 0,Y 202.264,Z 594.482,A -85,B 0,C 180,E1 -21661.461,E2 -21661.461} C_VEL
LIN {X 0,Y 198.5,Z 601.984,A -85,B 0,C 180,E1 -21664.859,E2 -21664.859} C_VEL
LIN {X 0,Y 195.118,Z 608.989,A -85,B 0,C 180,E1 -21668.889,E2 -21668.889} C_VEL
LIN {X 0,Y 192.702,Z 614.506,A -85,B 0,C 180,E1 -21673.037,E2 -21673.037} C_VEL
LIN {X 0,Y 191.077,Z 618.684,A -85,B 0,C 180,E1 -21677.251,E2 -21677.251} C_VEL
LIN {X 0,Y 190.327,Z 621.621,A -85,B 0,C 180,E1 -21681.506,E2 -21681.506} C_VEL
LIN {X 0,Y 190.083,Z 623.376,A -85,B 0,C 180,E1 -21685.759,E2 -21685.759} C_VEL
LIN {X 0,Y 190.264,Z 623.981,A -85,B 0,C 180,E1 -21690,E2 -21690} C_VEL
LIN {X 0,Y 190.081,Z 623.361,A -85,B 0,C 180,E1 -21694.241,E2 -21694.241} C_VEL
LIN {X 0,Y 190.286,Z 621.585,A -85,B 0,C 180,E1 -21698.495,E2 -21698.495} C_VEL
LIN {X 0,Y 191.072,Z 618.633,A -85,B 0,C 180,E1 -21702.749,E2 -21702.749} C_VEL
LIN {X 0,Y 192.662,Z 614.442,A -85,B 0,C 180,E1 -21706.967,E2 -21706.967} C_VEL
LIN {X 0,Y 195.097,Z 608.901,A -85,B 0,C 180,E1 -21711.114,E2 -21711.114} C_VEL
LIN {X 0,Y 198.518,Z 601.866,A -85,B 0,C 180,E1 -21715.139,E2 -21715.139} C_VEL
LIN {X 0,Y 202.278,Z 594.351,A -85,B 0,C 180,E1 -21718.537,E2 -21718.537} C_VEL
LIN {X 0,Y 206.49,Z 585.311,A -85,B 0,C 180,E1 -21721.83,E2 -21721.83} C_VEL
LIN {X 0,Y 210.731,Z 576.05,A -85,B 0,C 180,E1 -21724.537,E2 -21724.537} C_VEL
LIN {X 0,Y 215.454,Z 565.171,A -85,B 0,C 180,E1 -21727.117,E2 -21727.117} C_VEL
LIN {X 0,Y 220.229,Z 553.303,A -85,B 0,C 180,E1 -21729.363,E2 -21729.363} C_VEL
LIN {X 0,Y 224.879,Z 539.885,A -85,B 0,C 180,E1 -21731.405,E2 -21731.405} C_VEL
LIN {X 0,Y 229.099,Z 525.977,A -85,B 0,C 180,E1 -21733.042,E2 -21733.042} C_VEL
LIN {X 0,Y 232.671,Z 511.969,A -85,B 0,C 180,E1 -21734.306,E2 -21734.306} C_VEL
LIN {X 0,Y 235.698,Z 496.969,A -85,B 0,C 180,E1 -21735.312,E2 -21735.312} C_VEL
LIN {X 0,Y 237.928,Z 481.264,A -85,B 0,C 180,E1 -21736.052,E2 -21736.052} C_VEL
LIN {X 0,Y 239.594,Z 461.352,A -85,B 0,C 180,E1 -21736.626,E2 -21736.626} C_VEL
LIN {X 0,Y 243.776,Z 395.243,A -85,B 0,C 180,E1 -21738.389,E2 -21738.389} C_VEL
LIN {X 0,Y 238.099,Z 381.844,A -85,B 0,C 180,E1 -21740.555,E2 -21740.555} C_VEL
LIN {X 0,Y 231.628,Z 368.521,A -85,B 0,C 180,E1 -21743.193,E2 -21743.193} C_VEL
LIN {X 0,Y 224.449,Z 355.513,A -85,B 0,C 180,E1 -21746.422,E2 -21746.422} C_VEL
LIN {X 0,Y 218.256,Z 345.525,A -85,B 0,C 180,E1 -21749.559,E2 -21749.559} C_VEL
LIN {X 0,Y 214.874,Z 340.989,A -85,B 0,C 180,E1 -21751.423,E2 -21751.423} C_VEL
LIN {X 0,Y 211.854,Z 337.066,A -85,B 0,C 180,E1 -21753.231,E2 -21753.231} C_VEL
LIN {X 0,Y 208.342,Z 332.918,A -85,B 0,C 180,E1 -21755.526,E2 -21755.526} C_VEL
LIN {X 0,Y 207.367,Z 331.391,A -85,B 0,C 180,E1 -21756.246,E2 -21756.246} C_VEL
LIN {X 0,Y 204.697,Z 328.953,A -85,B 0,C 180,E1 -21758.209,E2 -21758.209} C_VEL
LIN {X 0,Y 202.974,Z 325.923,A -85,B 0,C 180,E1 -21759.742,E2 -21759.742} C_VEL
LIN {X 0,Y 200.291,Z 324.056,A -85,B 0,C 180,E1 -21762.117,E2 -21762.117} C_VEL
LIN {X 0,Y 198.543,Z 321.289,A -85,B 0,C 180,E1 -21764.078,E2 -21764.078} C_VEL
LIN {X 0,Y 198.193,Z 320.183,A -85,B 0,C 180,E1 -21764.577,E2 -21764.577} C_VEL
LIN {X 0,Y 195.088,Z 318.396,A -85,B 0,C 180,E1 -21768.572,E2 -21768.572} C_VEL
LIN {X 0,Y 193.288,Z 315.358,A -85,B 0,C 180,E1 -21772.295,E2 -21772.295} C_VEL
LIN {X 0,Y 192.953,Z 314.066,A -85,B 0,C 180,E1 -21773.596,E2 -21773.596} C_VEL
LIN {X 0,Y 193.224,Z 314.031,A -85,B 0,C 180,E1 -21777.916,E2 -21777.916} C_VEL
LIN {X 0,Y 193.406,Z 314.014,A -85,B 0,C 180,E1 -21780,E2 -21780} C_VEL
LIN {X 0,Y 192.937,Z 314.073,A -85,B 0,C 180,E1 -21784.178,E2 -21784.178} C_VEL
LIN {X 0,Y 192.966,Z 314.113,A -85,B 0,C 180,E1 -21787.061,E2 -21787.061} C_VEL
LIN {X 0,Y 194.027,Z 317.004,A -85,B 0,C 180,E1 -21789.95,E2 -21789.95} C_VEL
LIN {X 0,Y 196.17,Z 319.322,A -85,B 0,C 180,E1 -21793.466,E2 -21793.466} C_VEL
LIN {X 0,Y 198.244,Z 320.369,A -85,B 0,C 180,E1 -21795.947,E2 -21795.947} C_VEL
LIN {X 0,Y 199.628,Z 323.269,A -85,B 0,C 180,E1 -21797.647,E2 -21797.647} C_VEL
LIN {X 0,Y 201.924,Z 325.403,A -85,B 0,C 180,E1 -21799.838,E2 -21799.838} C_VEL
LIN {X 0,Y 203.106,Z 326.142,A -85,B 0,C 180,E1 -21800.826,E2 -21800.826} C_VEL
